KUKA KRL program: MyProgram_109().src

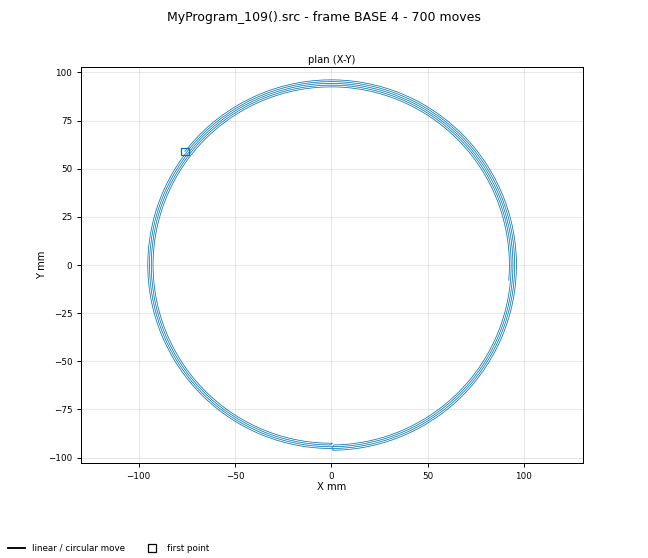
[picture p0: tool path of MyProgram_109().src in frame BASE 4, 700 of 700 moves have a stored position in this frame; points joined in program order, loops and branches not executed]
&ACCESS RVP
&REL 1
&PARAM TEMPLATE = C:\KRC\Roboter\Template\vorgabe
&PARAM EDITMASK = *
DEF MyProgram_109()
; ---- Setting reference (Base) ----
$BASE = BASE_DATA[4]

; --------------------------
; ---- Setting tool (TCP) ----
$TOOL = TOOL_DATA[3]
; --------------------------

$VEL.CP = VEL_APROX_PRINT
Startdeposition()
$VEL.CP = VEL_PRINT
LIN {X -75.9635,Y 58.9825,Z 96,A 136.7179,B 24.9196,C -2.0702,E1 24.8745,E2 -51.4268} C_DIS
LIN {X -71.624,Y 64.1816,Z 96,A 131.6242,B 24.9214,C -2.047,E1 24.884,E2 -46.2546} C_DIS
LIN {X -67.7687,Y 68.2403,Z 96,A 129.5352,B 24.9177,C -2.0948,E1 24.8879,E2 -44.2707} C_DIS
LIN {X -63.6529,Y 72.0961,Z 96,A 126.1542,B 24.9171,C -2.1019,E1 24.8948,E2 -40.8928} C_DIS
LIN {X -60.8353,Y 74.488,Z 96,A 123.6334,B 24.9176,C -2.0964,E1 24.9002,E2 -38.3493} C_DIS
LIN {X -56.4645,Y 77.852,Z 96,A 120.304,B 24.9171,C -2.1019,E1 24.9076,E2 -35.021} C_DIS
LIN {X -51.644,Y 81.1313,Z 96,A 116.9295,B 24.9164,C -2.1118,E1 24.9155,E2 -31.659} C_DIS
LIN {X -49.5866,Y 82.4052,Z 96,A 114.7873,B 24.918,C -2.0916,E1 24.9207,E2 -29.4622} C_DIS
LIN {X -45.8465,Y 84.5421,Z 96,A 112.8787,B 24.9159,C -2.1175,E1 24.9253,E2 -27.6098} C_DIS
LIN {X -39.8443,Y 87.5319,Z 96,A 108.9645,B 24.9152,C -2.1264,E1 24.9351,E2 -23.7067} C_DIS
LIN {X -36.8225,Y 88.8463,Z 96,A 106.6234,B 24.916,C -2.1167,E1 24.9412,E2 -21.337} C_DIS
LIN {X -32.9991,Y 90.3345,Z 96,A 104.4246,B 24.9151,C -2.1281,E1 24.9468,E2 -19.1608} C_DIS
LIN {X -29.4819,Y 91.5429,Z 96,A 101.6282,B 24.9164,C -2.1114,E1 24.9544,E2 -16.3196} C_DIS
LIN {X -25.5098,Y 92.7293,Z 96,A 100.0399,B 24.9138,C -2.1435,E1 24.9585,E2 -14.805} C_DIS
LIN {X -20.1495,Y 94.0393,Z 96,A 96.4801,B 24.9143,C -2.1373,E1 24.9682,E2 -11.2257} C_DIS
LIN {X -16.8432,Y 94.6869,Z 96,A 93.9105,B 24.9157,C -2.1199,E1 24.9754,E2 -8.6122} C_DIS
LIN {X -12.9376,Y 95.3007,Z 96,A 92.2981,B 24.9136,C -2.1465,E1 24.9797,E2 -7.0617} C_DIS
LIN {X -9.0125,Y 95.7501,Z 96,A 89.8172,B 24.9138,C -2.1435,E1 24.9866,E2 -4.5721} C_DIS
LIN {X -5.6055,Y 96.0101,Z 96,A 87.7986,B 24.9138,C -2.1449,E1 24.9922,E2 -2.5561} C_DIS
LIN {X -3.2117,Y 96.1198,Z 96,A 85.5461,B 24.9159,C -2.1171,E1 24.9987,E2 -0.2373} C_DIS
LIN {X 1.3526,Y 96.1645,Z 96,A 83.5892,B 24.9138,C -2.1437,E1 25.0039,E2 1.6563} C_DIS
LIN {X 4.7623,Y 96.0567,Z 96,A 81.5003,B 24.914,C -2.1419,E1 25.0098,E2 3.749} C_DIS
LIN {X 8.4191,Y 95.8048,Z 96,A 79.3633,B 24.9138,C -2.1434,E1 25.0157,E2 5.8814} C_DIS
LIN {X 11.8183,Y 95.4458,Z 96,A 77.2973,B 24.9139,C -2.142,E1 25.0214,E2 7.9492} C_DIS
LIN {X 15.3543,Y 94.9409,Z 96,A 75.1985,B 24.9139,C -2.1424,E1 25.0272,E2 10.045} C_DIS
LIN {X 19.7138,Y 94.1317,Z 96,A 72.7441,B 24.9135,C -2.1479,E1 25.0339,E2 12.4835} C_DIS
LIN {X 25.2917,Y 92.7882,Z 96,A 69.3515,B 24.9135,C -2.1468,E1 25.0431,E2 15.8737} C_DIS
LIN {X 29.6089,Y 91.5018,Z 96,A 66.6503,B 24.9138,C -2.1442,E1 25.0503,E2 18.5764} C_DIS
LIN {X 32.7031,Y 90.4425,Z 96,A 64.5541,B 24.9143,C -2.1372,E1 25.0559,E2 20.6849} C_DIS
LIN {X 35.084,Y 89.5455,Z 96,A 62.7776,B 24.9152,C -2.1264,E1 25.0606,E2 22.4831} C_DIS
LIN {X 40.332,Y 87.3079,Z 96,A 59.687,B 24.9146,C -2.1337,E1 25.0684,E2 25.5489} C_DIS
LIN {X 43.239,Y 85.9067,Z 96,A 57.7408,B 24.9149,C -2.1304,E1 25.0733,E2 27.4977} C_DIS
LIN {X 45.9132,Y 84.5059,Z 96,A 55.8586,B 24.9153,C -2.125,E1 25.0779,E2 29.3873} C_DIS
LIN {X 49.0395,Y 82.731,Z 96,A 53.7927,B 24.9153,C -2.1246,E1 25.0829,E2 31.4477} C_DIS
LIN {X 53.5705,Y 79.8712,Z 96,A 50.4819,B 24.9161,C -2.1153,E1 25.0907,E2 34.7699} C_DIS
LIN {X 56.5092,Y 77.8211,Z 96,A 48.2139,B 24.9168,C -2.1068,E1 25.0959,E2 37.0501} C_DIS
LIN {X 60.8788,Y 74.4528,Z 96,A 45.1605,B 24.9166,C -2.1093,E1 25.1025,E2 40.0861} C_DIS
LIN {X 66.2445,Y 69.7221,Z 96,A 40.9352,B 24.9171,C -2.1021,E1 25.1113,E2 44.3115} C_DIS
LIN {X 68.9933,Y 67.0025,Z 96,A 38.1075,B 24.919,C -2.0778,E1 25.1169,E2 47.1846} C_DIS
LIN {X 71.5664,Y 64.2459,Z 96,A 36.4875,B 24.9176,C -2.096,E1 25.1199,E2 48.7544} C_DIS
LIN {X 73.2967,Y 62.2647,Z 96,A 34.5911,B 24.9189,C -2.0801,E1 25.1234,E2 50.6797} C_DIS
LIN {X 75.914,Y 59.0468,Z 96,A 32.1059,B 24.9194,C -2.0737,E1 25.1277,E2 53.1686} C_DIS
LIN {X 78.5859,Y 55.4417,Z 96,A 29.6936,B 24.9191,C -2.0768,E1 25.1316,E2 55.5618} C_DIS
LIN {X 80.5905,Y 52.4835,Z 96,A 27.4533,B 24.9199,C -2.0671,E1 25.1351,E2 57.8137} C_DIS
LIN {X 82.391,Y 49.6099,Z 96,A 25.7028,B 24.9195,C -2.072,E1 25.1376,E2 59.5439} C_DIS
LIN {X 85.0356,Y 44.9247,Z 96,A 22.1086,B 24.9213,C -2.0486,E1 25.1425,E2 63.1744} C_DIS
LIN {X 87.1678,Y 40.6331,Z 96,A 19.8069,B 24.9203,C -2.0615,E1 25.1452,E2 65.4332} C_DIS
LIN {X 89.0887,Y 36.2281,Z 96,A 16.8208,B 24.9213,C -2.0486,E1 25.1485,E2 68.4335} C_DIS
LIN {X 90.7833,Y 31.7437,Z 96,A 13.9291,B 24.9221,C -2.0388,E1 25.1513,E2 71.3321} C_DIS
LIN {X 92.5603,Y 26.1125,Z 96,A 10.452,B 24.9227,C -2.0298,E1 25.1542,E2 74.8108} C_DIS
LIN {X 93.3092,Y 23.301,Z 96,A 8.1375,B 24.9248,C -2.0023,E1 25.1558,E2 77.1767} C_DIS
LIN {X 94.1518,Y 19.6159,Z 96,A 6.4875,B 24.9236,C -2.0183,E1 25.1567,E2 78.7795} C_DIS
LIN {X 94.8044,Y 16.171,Z 96,A 4.4178,B 24.9241,C -2.0125,E1 25.1577,E2 80.8507} C_DIS
LIN {X 95.3297,Y 12.7141,Z 96,A 2.338,B 24.9245,C -2.006,E1 25.1586,E2 82.9335} C_DIS
LIN {X 95.7187,Y 9.3522,Z 96,A 0.2659,B 24.9252,C -1.9975,E1 25.1592,E2 85.0135} C_DIS
LIN {X 96.0088,Y 5.6288,Z 96,A -1.8781,B 24.9255,C -1.9935,E1 25.1596,E2 87.1542} C_DIS
LIN {X 96.1411,Y 2.5178,Z 96,A -3.7568,B 24.926,C -1.9866,E1 25.1598,E2 89.0379} C_DIS
LIN {X 96.1691,Y -0.9828,Z 96,A -5.8078,B 24.9264,C -1.9813,E1 25.1598,E2 91.0894} C_DIS
LIN {X 96.0512,Y -4.8615,Z 96,A -8.2755,B 24.9274,C -1.9678,E1 25.1595,E2 93.5741} C_DIS
LIN {X 95.7693,Y -8.8044,Z 96,A -10.4034,B 24.9274,C -1.969,E1 25.159,E2 95.6867} C_DIS
LIN {X 95.3701,Y -12.4021,Z 96,A -12.583,B 24.9279,C -1.9611,E1 25.1583,E2 97.8719} C_DIS
LIN {X 94.8345,Y -15.991,Z 96,A -14.5993,B 24.9279,C -1.9598,E1 25.1574,E2 99.8795} C_DIS
LIN {X 94.3756,Y -18.5099,Z 96,A -16.6489,B 24.9298,C -1.9348,E1 25.1563,E2 101.9762} C_DIS
LIN {X 93.7019,Y -21.6617,Z 96,A -18.0886,B 24.9289,C -1.9471,E1 25.1554,E2 103.3784} C_DIS
LIN {X 93.134,Y -23.986,Z 96,A -20.0266,B 24.9307,C -1.9229,E1 25.154,E2 105.3622} C_DIS
LIN {X 92.2114,Y -27.3189,Z 96,A -22.127,B 24.9313,C -1.9149,E1 25.1524,E2 107.4695} C_DIS
LIN {X 91.1057,Y -30.8062,Z 96,A -23.3453,B 24.9291,C -1.945,E1 25.1514,E2 108.61} C_DIS
LIN {X 89.8798,Y -34.2186,Z 96,A -26.3157,B 24.9318,C -1.9072,E1 25.1484,E2 111.653} C_DIS
LIN {X 88.6877,Y -37.1993,Z 96,A -28.0731,B 24.9318,C -1.9072,E1 25.1465,E2 113.4006} C_DIS
LIN {X 86.7733,Y -41.4693,Z 96,A -30.9801,B 24.9327,C -1.8943,E1 25.1431,E2 116.3224} C_DIS
LIN {X 85.3222,Y -44.3806,Z 96,A -32.8135,B 24.9329,C -1.8925,E1 25.1408,E2 118.1503} C_DIS
LIN {X 81.7409,Y -50.6735,Z 96,A -36.7914,B 24.9329,C -1.8929,E1 25.1352,E2 122.1068} C_DIS
LIN {X 79.0751,Y -54.7396,Z 96,A -39.9312,B 24.9341,C -1.8755,E1 25.1303,E2 125.2721} C_DIS
LIN {X 75.347,Y -59.7672,Z 96,A -43.4414,B 24.9341,C -1.8738,E1 25.1243,E2 128.7697} C_DIS
LIN {X 73.0047,Y -62.6074,Z 96,A -45.4134,B 24.934,C -1.8765,E1 25.1208,E2 130.7263} C_DIS
LIN {X 70.1761,Y -65.7618,Z 96,A -48.3985,B 24.9357,C -1.8527,E1 25.1151,E2 133.7545} C_DIS
LIN {X 66.9268,Y -69.0661,Z 96,A -50.7849,B 24.9351,C -1.8601,E1 25.1105,E2 136.1133} C_DIS
LIN {X 64.5588,Y -71.2861,Z 96,A -52.5649,B 24.9351,C -1.8613,E1 25.1068,E2 137.8831} C_DIS
LIN {X 61.8693,Y -73.6324,Z 96,A -55.2908,B 24.937,C -1.834,E1 25.1009,E2 140.663} C_DIS
LIN {X 59.3273,Y -75.6948,Z 96,A -56.8127,B 24.9361,C -1.8458,E1 25.0977,E2 142.1513} C_DIS
LIN {X 56.7069,Y -77.6763,Z 96,A -58.7892,B 24.9365,C -1.841,E1 25.0932,E2 144.1322} C_DIS
LIN {X 54.6408,Y -79.1438,Z 96,A -60.489,B 24.9372,C -1.8308,E1 25.0893,E2 145.8502} C_DIS
LIN {X 48.4141,Y -83.1004,Z 96,A -64.6992,B 24.9372,C -1.8294,E1 25.0793,E2 150.0504} C_DIS
LIN {X 43.3453,Y -85.8526,Z 96,A -68.4345,B 24.9384,C -1.8125,E1 25.07,E2 153.8152} C_DIS
LIN {X 38.7385,Y -88.0268,Z 96,A -70.8505,B 24.9372,C -1.8306,E1 25.064,E2 156.1822} C_DIS
LIN {X 36.2891,Y -89.0639,Z 96,A -72.9477,B 24.9386,C -1.8095,E1 25.0585,E2 158.3245} C_DIS
LIN {X 32.3499,Y -90.5704,Z 96,A -76.1015,B 24.9404,C -1.7829,E1 25.0501,E2 161.5346} C_DIS
LIN {X 27.4941,Y -92.1595,Z 96,A -77.8804,B 24.9376,C -1.8253,E1 25.0456,E2 163.2102} C_DIS
LIN {X 22.4848,Y -93.5083,Z 96,A -81.358,B 24.9387,C -1.8079,E1 25.0361,E2 166.7234} C_DIS
LIN {X 17.5814,Y -94.5541,Z 96,A -84.3174,B 24.9388,C -1.8063,E1 25.028,E2 169.6831} C_DIS
LIN {X 14.1878,Y -95.1222,Z 96,A -86.3586,B 24.9389,C -1.8051,E1 25.0223,E2 171.725} C_DIS
LIN {X 10.552,Y -95.594,Z 96,A -88.5213,B 24.9389,C -1.8045,E1 25.0163,E2 173.8875} C_DIS
LIN {X 7.0264,Y -95.9176,Z 96,A -90.6506,B 24.9391,C -1.8028,E1 25.0104,E2 176.0198} C_DIS
LIN {X 3.4991,Y -96.111,Z 96,A -92.7507,B 24.9391,C -1.8022,E1 25.0046,E2 178.1207} C_DIS
LIN {X 0.6665,Y -96.1682,Z 96,A -93.7382,B 24.9374,C -1.8268,E1 25.002,E2 179.0497} C_DIS
Enddeposition()
LIN {X 0.6665,Y -96.1682,Z 96,A -93.7382,B 24.9374,C -1.8268,E1 25.002,E2 179.0497} C_DIS
Startdeposition()
$VEL.CP = VEL_PRINT
LIN {X 1.0872,Y -95.2543,Z 96,A -93.1803,B 24.9356,C -1.8535,E1 25.0037,E2 178.4284} C_DIS
LIN {X 4.3828,Y -95.1587,Z 96,A -91.1856,B 24.9356,C -1.8547,E1 25.0093,E2 176.4315} C_DIS
LIN {X 7.8747,Y -94.9336,Z 96,A -89.0988,B 24.9355,C -1.855,E1 25.0151,E2 174.3449} C_DIS
LIN {X 11.567,Y -94.5556,Z 96,A -86.7396,B 24.9351,C -1.8609,E1 25.0217,E2 171.9734} C_DIS
LIN {X 15.6874,Y -93.9586,Z 96,A -84.4427,B 24.9355,C -1.8552,E1 25.028,E2 169.6922} C_DIS
LIN {X 21.2338,Y -92.8627,Z 96,A -81.221,B 24.9357,C -1.8516,E1 25.0367,E2 166.483} C_DIS
LIN {X 24.7928,Y -91.9762,Z 96,A -78.7965,B 24.935,C -1.8619,E1 25.0433,E2 164.038} C_DIS
LIN {X 28.3124,Y -90.9545,Z 96,A -76.1297,B 24.9336,C -1.8815,E1 25.0506,E2 161.3294} C_DIS
LIN {X 31.5787,Y -89.8727,Z 96,A -74.2994,B 24.9341,C -1.8753,E1 25.0554,E2 159.5176} C_DIS
LIN {X 37.2004,Y -87.6954,Z 96,A -71.1813,B 24.935,C -1.8615,E1 25.0633,E2 156.439} C_DIS
LIN {X 39.5771,Y -86.6498,Z 96,A -69.4286,B 24.9344,C -1.871,E1 25.0679,E2 154.6683} C_DIS
LIN {X 42.7302,Y -85.1391,Z 96,A -66.5179,B 24.932,C -1.9047,E1 25.0753,E2 151.6857} C_DIS
LIN {X 46.6327,Y -83.0647,Z 96,A -64.7132,B 24.9339,C -1.8773,E1 25.0796,E2 149.9511} C_DIS
LIN {X 49.7001,Y -81.2667,Z 96,A -62.137,B 24.9325,C -1.8977,E1 25.0858,E2 147.3347} C_DIS
LIN {X 55.4137,Y -77.4831,Z 96,A -58.4667,B 24.9331,C -1.8888,E1 25.0942,E2 143.6976} C_DIS
LIN {X 58.1709,Y -75.4351,Z 96,A -55.6801,B 24.9308,C -1.9206,E1 25.1005,E2 140.8461} C_DIS
LIN {X 61.4032,Y -72.8299,Z 96,A -53.3642,B 24.9309,C -1.9193,E1 25.1054,E2 138.5423} C_DIS
LIN {X 64.027,Y -70.5345,Z 96,A -51.9557,B 24.9325,C -1.8979,E1 25.1083,E2 137.1899} C_DIS
LIN {X 65.8828,Y -68.8031,Z 96,A -50.2594,B 24.9318,C -1.908,E1 25.1117,E2 135.4768} C_DIS
LIN {X 69.6881,Y -64.9467,Z 96,A -46.334,B 24.9293,C -1.9416,E1 25.1194,E2 131.489} C_DIS
LIN {X 72.4219,Y -61.8822,Z 96,A -44.6671,B 24.9311,C -1.9171,E1 25.1224,E2 129.8874} C_DIS
LIN {X 74.3382,Y -59.5687,Z 96,A -41.9522,B 24.9282,C -1.9569,E1 25.1273,E2 127.0913} C_DIS
LIN {X 77.1265,Y -55.9108,Z 96,A -39.576,B 24.9288,C -1.9493,E1 25.1311,E2 124.7444} C_DIS
LIN {X 80.3004,Y -51.2466,Z 96,A -36.6114,B 24.9293,C -1.9423,E1 25.1356,E2 121.8112} C_DIS
LIN {X 83.327,Y -46.163,Z 96,A -33.0482,B 24.9285,C -1.9527,E1 25.1406,E2 118.2418} C_DIS
LIN {X 85.4364,Y -42.1302,Z 96,A -30.4276,B 24.9282,C -1.9563,E1 25.144,E2 115.6265} C_DIS
LIN {X 87.4708,Y -37.7268,Z 96,A -27.6993,B 24.9282,C -1.9578,E1 25.1471,E2 112.9095} C_DIS
LIN {X 89.7057,Y -32.0544,Z 96,A -23.7893,B 24.9266,C -1.9784,E1 25.1511,E2 108.9726} C_DIS
LIN {X 90.7958,Y -28.8219,Z 96,A -20.9247,B 24.9238,C -2.0165,E1 25.1535,E2 106.0343} C_DIS
LIN {X 92.1449,Y -24.163,Z 96,A -19.1061,B 24.9263,C -1.9829,E1 25.1548,E2 104.3054} C_DIS
LIN {X 92.8385,Y -21.3386,Z 96,A -16.7169,B 24.924,C -2.0134,E1 25.1564,E2 101.8583} C_DIS
LIN {X 93.524,Y -18.0992,Z 96,A -15.4794,B 24.9257,C -1.9905,E1 25.157,E2 100.6821} C_DIS
LIN {X 93.95,Y -15.7388,Z 96,A -13.7684,B 24.9246,C -2.0055,E1 25.1578,E2 98.9457} C_DIS
LIN {X 94.4624,Y -12.2949,Z 96,A -11.7086,B 24.9242,C -2.0109,E1 25.1586,E2 96.8854} C_DIS
LIN {X 94.8478,Y -8.8439,Z 96,A -9.6239,B 24.9237,C -2.0174,E1 25.1592,E2 94.7975} C_DIS
LIN {X 95.1282,Y -4.9993,Z 96,A -7.3977,B 24.9234,C -2.0213,E1 25.1596,E2 92.5753} C_DIS
LIN {X 95.2462,Y -1.5801,Z 96,A -5.2259,B 24.9225,C -2.0324,E1 25.1598,E2 90.3904} C_DIS
LIN {X 95.2392,Y 1.9593,Z 96,A -3.1527,B 24.9222,C -2.037,E1 25.1598,E2 88.3184} C_DIS
LIN {X 95.1078,Y 5.3688,Z 96,A -1.1401,B 24.9218,C -2.0421,E1 25.1594,E2 86.3059} C_DIS
LIN {X 94.8541,Y 8.7756,Z 96,A 0.9363,B 24.9212,C -2.0495,E1 25.159,E2 84.2244} C_DIS
LIN {X 94.4613,Y 12.3033,Z 96,A 3.0514,B 24.9208,C -2.0555,E1 25.1583,E2 82.1077} C_DIS
LIN {X 93.918,Y 15.9302,Z 96,A 5.3098,B 24.9201,C -2.0644,E1 25.1573,E2 79.8414} C_DIS
LIN {X 93.2612,Y 19.4094,Z 96,A 8.2612,B 24.9171,C -2.1029,E1 25.1556,E2 76.8164} C_DIS
LIN {X 92.1175,Y 24.2694,Z 96,A 10.2054,B 24.9196,C -2.0711,E1 25.1543,E2 74.9585} C_DIS
LIN {X 91.0329,Y 28.0596,Z 96,A 12.9347,B 24.9179,C -2.092,E1 25.1521,E2 72.1954} C_DIS
LIN {X 88.9459,Y 34.104,Z 96,A 16.6021,B 24.9176,C -2.0965,E1 25.1486,E2 68.538} C_DIS
LIN {X 87.6252,Y 37.3672,Z 96,A 18.876,B 24.9166,C -2.1086,E1 25.1462,E2 66.248} C_DIS
LIN {X 85.6149,Y 41.7698,Z 96,A 22.096,B 24.915,C -2.1286,E1 25.1423,E2 62.9981} C_DIS
LIN {X 83.9203,Y 45.076,Z 96,A 23.6557,B 24.9166,C -2.1089,E1 25.1403,E2 61.4931} C_DIS
LIN {X 81.7775,Y 48.8564,Z 96,A 26.1789,B 24.9163,C -2.1125,E1 25.1368,E2 58.9744} C_DIS
LIN {X 80.3931,Y 51.1021,Z 96,A 28.2852,B 24.9144,C -2.1364,E1 25.1336,E2 56.8225} C_DIS
LIN {X 77.954,Y 54.7513,Z 96,A 30.614,B 24.9148,C -2.1312,E1 25.1299,E2 54.5172} C_DIS
LIN {X 74.8472,Y 58.9257,Z 96,A 34.1679,B 24.9129,C -2.1549,E1 25.1238,E2 50.9243} C_DIS
LIN {X 72.6176,Y 61.6524,Z 96,A 35.6693,B 24.9144,C -2.1365,E1 25.1212,E2 49.4731} C_DIS
LIN {X 70.5715,Y 63.9867,Z 96,A 38.272,B 24.9118,C -2.1684,E1 25.1162,E2 46.8066} C_DIS
LIN {X 67.8593,Y 66.8538,Z 96,A 39.8824,B 24.9137,C -2.1449,E1 25.1132,E2 45.2587} C_DIS
LIN {X 65.328,Y 69.3294,Z 96,A 42.9783,B 24.9104,C -2.1855,E1 25.1068,E2 42.0795} C_DIS
LIN {X 61.7288,Y 72.5525,Z 96,A 44.9914,B 24.9127,C -2.1577,E1 25.1027,E2 40.14} C_DIS
LIN {X 58.2198,Y 75.3975,Z 96,A 47.2958,B 24.9135,C -2.1475,E1 25.0977,E2 37.8685} C_DIS
LIN {X 55.7027,Y 77.277,Z 96,A 49.5726,B 24.9121,C -2.165,E1 25.0925,E2 35.5583} C_DIS
LIN {X 50.921,Y 80.5087,Z 96,A 52.8806,B 24.9121,C -2.1646,E1 25.0849,E2 32.2624} C_DIS
LIN {X 47.3722,Y 82.645,Z 96,A 55.4654,B 24.9115,C -2.1717,E1 25.0786,E2 29.6687} C_DIS
LIN {X 44.2239,Y 84.3717,Z 96,A 57.403,B 24.912,C -2.1665,E1 25.0739,E2 27.749} C_DIS
LIN {X 42.1748,Y 85.4144,Z 96,A 59.1206,B 24.9108,C -2.1804,E1 25.0695,E2 26.0031} C_DIS
LIN {X 38.4057,Y 87.1748,Z 96,A 62.1578,B 24.909,C -2.2027,E1 25.0617,E2 22.9206} C_DIS
LIN {X 34.9011,Y 88.6354,Z 96,A 63.5697,B 24.9114,C -2.1735,E1 25.0582,E2 21.5811} C_DIS
LIN {X 32.6409,Y 89.4923,Z 96,A 65.2605,B 24.9106,C -2.1834,E1 25.0537,E2 19.8705} C_DIS
LIN {X 28.8125,Y 90.7989,Z 96,A 68.2218,B 24.9089,C -2.2043,E1 25.0458,E2 16.8652} C_DIS
LIN {X 25.4772,Y 91.7904,Z 96,A 69.6449,B 24.9107,C -2.1817,E1 25.0421,E2 15.4979} C_DIS
LIN {X 23.1402,Y 92.4072,Z 96,A 71.7537,B 24.9087,C -2.206,E1 25.0362,E2 13.3348} C_DIS
LIN {X 19.7611,Y 93.1886,Z 96,A 73.6606,B 24.9092,C -2.2006,E1 25.0311,E2 11.4432} C_DIS
LIN {X 16.0236,Y 93.9024,Z 96,A 75.5551,B 24.9102,C -2.1875,E1 25.026,E2 9.5818} C_DIS
LIN {X 13.1162,Y 94.3523,Z 96,A 77.4705,B 24.9098,C -2.1931,E1 25.0206,E2 7.6548} C_DIS
LIN {X 9.6502,Y 94.7695,Z 96,A 79.4669,B 24.9101,C -2.1898,E1 25.0151,E2 5.6677} C_DIS
LIN {X 6.4585,Y 95.04,Z 96,A 81.3482,B 24.9101,C -2.1883,E1 25.0099,E2 3.7908} C_DIS
LIN {X 3.128,Y 95.208,Z 96,A 83.3988,B 24.9101,C -2.1898,E1 25.0042,E2 1.7374} C_DIS
LIN {X -0.1984,Y 95.2593,Z 96,A 85.7914,B 24.909,C -2.203,E1 24.9974,E2 -0.6866} C_DIS
LIN {X -5.0768,Y 95.124,Z 96,A 88.3402,B 24.9101,C -2.1887,E1 24.9904,E2 -3.2017} C_DIS
LIN {X -8.2975,Y 94.8982,Z 96,A 91.1194,B 24.9078,C -2.2168,E1 24.9825,E2 -6.0491} C_DIS
LIN {X -12.8562,Y 94.3892,Z 96,A 92.9174,B 24.9107,C -2.1819,E1 24.9777,E2 -7.7656} C_DIS
LIN {X -18.277,Y 93.4898,Z 96,A 96.3114,B 24.9107,C -2.1825,E1 24.9684,E2 -11.1642} C_DIS
LIN {X -22.9547,Y 92.4528,Z 96,A 99.344,B 24.9105,C -2.1849,E1 24.9601,E2 -14.2066} C_DIS
LIN {X -25.6453,Y 91.7428,Z 96,A 101.5323,B 24.9092,C -2.2007,E1 24.9541,E2 -16.4359} C_DIS
LIN {X -29.2113,Y 90.6699,Z 96,A 102.9294,B 24.9117,C -2.1696,E1 24.9506,E2 -17.7615} C_DIS
LIN {X -31.5975,Y 89.8661,Z 96,A 104.6823,B 24.9112,C -2.1757,E1 24.9459,E2 -19.5324} C_DIS
LIN {X -34.6764,Y 88.7237,Z 96,A 106.9992,B 24.9105,C -2.1846,E1 24.9398,E2 -21.8752} C_DIS
LIN {X -38.9999,Y 86.91,Z 96,A 110.3805,B 24.9093,C -2.1994,E1 24.931,E2 -25.2997} C_DIS
LIN {X -43.2642,Y 84.8677,Z 96,A 112.3516,B 24.912,C -2.1655,E1 24.9263,E2 -27.1955} C_DIS
LIN {X -48.942,Y 81.7269,Z 96,A 116.0651,B 24.9131,C -2.1524,E1 24.9173,E2 -30.8885} C_DIS
LIN {X -51.9423,Y 79.8527,Z 96,A 118.6277,B 24.9123,C -2.1627,E1 24.9112,E2 -33.4839} C_DIS
LIN {X -57.0114,Y 76.3154,Z 96,A 122.1932,B 24.9133,C -2.1501,E1 24.9031,E2 -37.0318} C_DIS
LIN {X -59.6988,Y 74.2327,Z 96,A 124.9562,B 24.9117,C -2.1693,E1 24.897,E2 -39.8509} C_DIS
LIN {X -62.9852,Y 71.4658,Z 96,A 127.6584,B 24.9119,C -2.1674,E1 24.8913,E2 -42.5592} C_DIS
LIN {X -66.4029,Y 68.3018,Z 96,A 129.6912,B 24.9145,C -2.1355,E1 24.8873,E2 -44.5245} C_DIS
LIN {X -71.0089,Y 63.4984,Z 96,A 134.2396,B 24.9138,C -2.1434,E1 24.8786,E2 -49.1115} C_DIS
LIN {X -73.4528,Y 60.6554,Z 96,A 135.7348,B 24.9163,C -2.1129,E1 24.8761,E2 -50.5409} C_DIS
LIN {X -74.9969,Y 58.7363,Z 96,A 137.5717,B 24.9157,C -2.1204,E1 24.8728,E2 -52.4044} C_DIS
LIN {X -77.9953,Y 54.6919,Z 96,A 140.4948,B 24.9166,C -2.1088,E1 24.8681,E2 -55.314} C_DIS
LIN {X -80.3638,Y 51.1478,Z 96,A 142.9077,B 24.9175,C -2.0968,E1 24.8644,E2 -57.7104} C_DIS
LIN {X -81.5228,Y 49.2788,Z 96,A 144.8947,B 24.9162,C -2.1144,E1 24.8615,E2 -59.7496} C_DIS
LIN {X -83.282,Y 46.2435,Z 96,A 146.3012,B 24.9184,C -2.0857,E1 24.8596,E2 -61.095} C_DIS
LIN {X -85.6489,Y 41.6961,Z 96,A 149.6025,B 24.9186,C -2.0835,E1 24.8554,E2 -64.4088} C_DIS
LIN {X -87.122,Y 38.5268,Z 96,A 152.1913,B 24.9179,C -2.0927,E1 24.8524,E2 -67.0339} C_DIS
LIN {X -88.4184,Y 35.4506,Z 96,A 153.7568,B 24.9195,C -2.0725,E1 24.8508,E2 -68.5596} C_DIS
LIN {X -89.9884,Y 31.2488,Z 96,A 156.3114,B 24.9205,C -2.0596,E1 24.8484,E2 -71.098} C_DIS
LIN {X -90.9272,Y 28.4006,Z 96,A 158.8014,B 24.9192,C -2.0759,E1 24.8462,E2 -73.6411} C_DIS
LIN {X -91.9184,Y 25.007,Z 96,A 160.8116,B 24.92,C -2.0654,E1 24.8448,E2 -75.6381} C_DIS
LIN {X -92.8299,Y 21.3756,Z 96,A 163.0358,B 24.9206,C -2.0574,E1 24.8434,E2 -77.8562} C_DIS
LIN {X -94.0127,Y 15.3638,Z 96,A 167.6057,B 24.9193,C -2.0741,E1 24.8412,E2 -82.4931} C_DIS
LIN {X -94.7949,Y 9.4075,Z 96,A 169.84,B 24.9236,C -2.0182,E1 24.8405,E2 -84.6074} C_DIS
LIN {X -95.1699,Y 4.1221,Z 96,A 173.7598,B 24.9226,C -2.0313,E1 24.8398,E2 -88.582} C_DIS
LIN {X -95.2578,Y 0.6008,Z 96,A 175.2863,B 24.9246,C -2.0056,E1 24.8398,E2 -90.0563} C_DIS
LIN {X -95.2219,Y -2.6748,Z 96,A 177.9803,B 24.9233,C -2.0224,E1 24.84,E2 -92.8067} C_DIS
LIN {X -95.036,Y -6.5179,Z 96,A -179.7635,B 24.924,C -2.0132,E1 24.8404,E2 -95.0544} C_DIS
LIN {X -94.7217,Y -10.1067,Z 96,A -178.3175,B 24.9263,C -1.9832,E1 24.8408,E2 -96.4376} C_DIS
LIN {X -94.3898,Y -12.8522,Z 96,A -175.5181,B 24.9239,C -2.0144,E1 24.8419,E2 -99.3283} C_DIS
LIN {X -93.5955,Y -17.7279,Z 96,A -172.6319,B 24.9248,C -2.0024,E1 24.8434,E2 -102.2029} C_DIS
LIN {X -92.6273,Y -22.2399,Z 96,A -170.6522,B 24.9274,C -1.9682,E1 24.8446,E2 -104.1125} C_DIS
LIN {X -91.7533,Y -25.6082,Z 96,A -167.8083,B 24.926,C -1.9861,E1 24.8468,E2 -107.0156} C_DIS
LIN {X -90.4912,Y -29.7636,Z 96,A -166.119,B 24.9288,C -1.9485,E1 24.8481,E2 -108.6248} C_DIS
LIN {X -89.0865,Y -33.7328,Z 96,A -162.7865,B 24.9275,C -1.9669,E1 24.8514,E2 -112.02} C_DIS
LIN {X -87.6764,Y -37.2455,Z 96,A -161.1154,B 24.9294,C -1.9407,E1 24.8531,E2 -113.6379} C_DIS
LIN {X -86.8228,Y -39.1933,Z 96,A -159.4056,B 24.9286,C -1.951,E1 24.8551,E2 -115.3817} C_DIS
LIN {X -83.3712,Y -46.0839,Z 96,A -155.3646,B 24.931,C -1.9189,E1 24.8602,E2 -119.3677} C_DIS
LIN {X -81.4344,Y -49.4242,Z 96,A -152.8186,B 24.9309,C -1.92,E1 24.8639,E2 -121.9295} C_DIS
LIN {X -80.0366,Y -51.6576,Z 96,A -151.1272,B 24.9309,C -1.9194,E1 24.8664,E2 -123.6279} C_DIS
LIN {X -77.5633,Y -55.3014,Z 96,A -148.2247,B 24.9309,C -1.921,E1 24.8711,E2 -126.5488} C_DIS
LIN {X -74.8125,Y -58.9695,Z 96,A -145.887,B 24.9323,C -1.9006,E1 24.875,E2 -128.8488} C_DIS
LIN {X -73.1049,Y -61.0741,Z 96,A -143.2197,B 24.9301,C -1.9312,E1 24.8799,E2 -131.6012} C_DIS
LIN {X -69.8305,Y -64.7943,Z 96,A -141.0485,B 24.9325,C -1.8975,E1 24.8839,E2 -133.7019} C_DIS
LIN {X -67.4187,Y -67.2999,Z 96,A -138.4075,B 24.9315,C -1.9114,E1 24.8892,E2 -136.3872} C_DIS
LIN {X -64.6426,Y -69.9696,Z 96,A -136.9837,B 24.934,C -1.8769,E1 24.8919,E2 -137.7347} C_DIS
LIN {X -60.9411,Y -73.2154,Z 96,A -133.7522,B 24.9337,C -1.8802,E1 24.8988,E2 -140.9866} C_DIS
LIN {X -57.9716,Y -75.5887,Z 96,A -131.5799,B 24.9343,C -1.8722,E1 24.9035,E2 -143.148} C_DIS
LIN {X -54.2195,Y -78.3236,Z 96,A -128.301,B 24.9335,C -1.8839,E1 24.9111,E2 -146.466} C_DIS
LIN {X -50.7684,Y -80.604,Z 96,A -126.153,B 24.9346,C -1.8685,E1 24.916,E2 -148.5843} C_DIS
LIN {X -48.1602,Y -82.189,Z 96,A -124.2715,B 24.9346,C -1.8674,E1 24.9206,E2 -150.469} C_DIS
LIN {X -44.9607,Y -83.9829,Z 96,A -122.0378,B 24.9348,C -1.8654,E1 24.926,E2 -152.7041} C_DIS
LIN {X -41.7501,Y -85.6225,Z 96,A -119.1409,B 24.9332,C -1.8878,E1 24.9335,E2 -155.6621} C_DIS
LIN {X -37.7165,Y -87.4753,Z 96,A -117.6159,B 24.9362,C -1.8455,E1 24.9371,E2 -157.09} C_DIS
LIN {X -34.2101,Y -88.9057,Z 96,A -114.6795,B 24.9347,C -1.8659,E1 24.9449,E2 -160.0813} C_DIS
LIN {X -28.2689,Y -90.968,Z 96,A -111.1811,B 24.9356,C -1.853,E1 24.9541,E2 -163.5556} C_DIS
LIN {X -23.0396,Y -92.4322,Z 96,A -107.6202,B 24.9351,C -1.8612,E1 24.9637,E2 -167.1416} C_DIS
LIN {X -19.7403,Y -93.1931,Z 96,A -105.8008,B 24.9357,C -1.8527,E1 24.9686,E2 -168.9428} C_DIS
LIN {X -16.418,Y -93.8348,Z 96,A -103.7725,B 24.9357,C -1.8517,E1 24.9742,E2 -170.971} C_DIS
LIN {X -13.1715,Y -94.3444,Z 96,A -101.7508,B 24.9357,C -1.8528,E1 24.9798,E2 -172.9971} C_DIS
LIN {X -9.6435,Y -94.7702,Z 96,A -99.6109,B 24.9357,C -1.8527,E1 24.9857,E2 -175.1378} C_DIS
LIN {X -5.8991,Y -95.0778,Z 96,A -97.3638,B 24.9357,C -1.8522,E1 24.992,E2 -177.3847} C_DIS
LIN {X -2.4876,Y -95.2277,Z 96,A -95.3064,B 24.9357,C -1.8526,E1 24.9978,E2 -179.4433} C_DIS
LIN {X 0.6651,Y -95.2549,Z 96,A -94.235,B 24.9377,C -1.8237,E1 25.0006,E2 -180.4464} C_DIS
Enddeposition()
LIN {X 0.6651,Y -95.2549,Z 96,A -94.235,B 24.9377,C -1.8237,E1 25.0006,E2 -180.4464} C_DIS
Startdeposition()
$VEL.CP = VEL_PRINT
LIN {X 0.2729,Y -94.3453,Z 96,A -94.7204,B 24.9372,C -1.831,E1 24.9993,E2 -179.9782} C_DIS
LIN {X -3.2853,Y -94.2888,Z 96,A -96.8702,B 24.9372,C -1.8311,E1 24.9932,E2 -177.8283} C_DIS
LIN {X -6.522,Y -94.1197,Z 96,A -98.8771,B 24.9372,C -1.8297,E1 24.9876,E2 -175.8176} C_DIS
LIN {X -9.9655,Y -93.8175,Z 96,A -100.9241,B 24.9372,C -1.8317,E1 24.982,E2 -173.7741} C_DIS
LIN {X -13.2272,Y -93.4134,Z 96,A -102.8791,B 24.937,C -1.8335,E1 24.9766,E2 -171.8219} C_DIS
LIN {X -16.7128,Y -92.8531,Z 96,A -105.0154,B 24.937,C -1.8344,E1 24.9707,E2 -169.6858} C_DIS
LIN {X -21.4523,Y -91.8742,Z 96,A -107.8471,B 24.9366,C -1.8394,E1 24.963,E2 -166.8624} C_DIS
LIN {X -24.0799,Y -91.2212,Z 96,A -109.7685,B 24.9372,C -1.8309,E1 24.9577,E2 -164.9181} C_DIS
LIN {X -27.8238,Y -90.1492,Z 96,A -111.8106,B 24.9363,C -1.8435,E1 24.9523,E2 -162.9025} C_DIS
LIN {X -31.0447,Y -89.0915,Z 96,A -114.169,B 24.9369,C -1.835,E1 24.946,E2 -160.5196} C_DIS
LIN {X -34.5678,Y -87.7844,Z 96,A -116.2895,B 24.9364,C -1.8426,E1 24.9405,E2 -158.4125} C_DIS
LIN {X -37.4941,Y -86.5752,Z 96,A -119.4711,B 24.9391,C -1.8031,E1 24.9321,E2 -155.1296} C_DIS
LIN {X -42.8069,Y -84.075,Z 96,A -122.2947,B 24.9371,C -1.8317,E1 24.9252,E2 -152.3666} C_DIS
LIN {X -45.6701,Y -82.5554,Z 96,A -123.7498,B 24.9358,C -1.8513,E1 24.9217,E2 -150.9538} C_DIS
LIN {X -48.2436,Y -81.0781,Z 96,A -125.5343,B 24.9355,C -1.8544,E1 24.9174,E2 -149.1714} C_DIS
LIN {X -51.4978,Y -79.0523,Z 96,A -128.5673,B 24.9369,C -1.8349,E1 24.9102,E2 -146.0824} C_DIS
LIN {X -54.5606,Y -76.9691,Z 96,A -130.4376,B 24.9358,C -1.851,E1 24.906,E2 -144.2439} C_DIS
LIN {X -58.058,Y -74.368,Z 96,A -132.9719,B 24.9352,C -1.8593,E1 24.9004,E2 -141.7201} C_DIS
LIN {X -60.7096,Y -72.2194,Z 96,A -135.0933,B 24.935,C -1.8616,E1 24.8958,E2 -139.5962} C_DIS
LIN {X -63.6332,Y -69.6554,Z 96,A -137.7244,B 24.9353,C -1.8576,E1 24.8903,E2 -136.9451} C_DIS
LIN {X -67.1546,Y -66.2668,Z 96,A -140.2784,B 24.9339,C -1.8771,E1 24.8853,E2 -134.4268} C_DIS
LIN {X -69.4973,Y -63.8055,Z 96,A -142.1591,B 24.9332,C -1.8875,E1 24.8817,E2 -132.5627} C_DIS
LIN {X -72.2652,Y -60.6546,Z 96,A -144.9903,B 24.9334,C -1.8842,E1 24.8765,E2 -129.7107} C_DIS
LIN {X -74.0205,Y -58.4977,Z 96,A -146.5759,B 24.9329,C -1.8915,E1 24.8738,E2 -128.135} C_DIS
LIN {X -77.4194,Y -53.9191,Z 96,A -150.2303,B 24.9328,C -1.8939,E1 24.8677,E2 -124.4687} C_DIS
LIN {X -79.4607,Y -50.8628,Z 96,A -152.4591,B 24.9323,C -1.8998,E1 24.8643,E2 -122.2426} C_DIS
LIN {X -81.3228,Y -47.8296,Z 96,A -154.5928,B 24.9319,C -1.9063,E1 24.8613,E2 -120.1136} C_DIS
LIN {X -82.7029,Y -45.4035,Z 96,A -157.4464,B 24.9341,C -1.8749,E1 24.8574,E2 -117.17} C_DIS
LIN {X -85.3496,Y -40.2077,Z 96,A -159.8606,B 24.9309,C -1.9197,E1 24.8545,E2 -114.8496} C_DIS
LIN {X -86.6279,Y -37.3732,Z 96,A -162.4683,B 24.9321,C -1.9028,E1 24.8516,E2 -112.187} C_DIS
LIN {X -88.2211,Y -33.4373,Z 96,A -164.2954,B 24.9299,C -1.9336,E1 24.8498,E2 -110.4232} C_DIS
LIN {X -89.4073,Y -30.1223,Z 96,A -166.2901,B 24.9291,C -1.9444,E1 24.848,E2 -108.4429} C_DIS
LIN {X -90.5858,Y -26.3716,Z 96,A -168.909,B 24.9291,C -1.9444,E1 24.8458,E2 -105.8088} C_DIS
LIN {X -91.411,Y -23.3468,Z 96,A -170.8034,B 24.9287,C -1.9504,E1 24.8445,E2 -103.918} C_DIS
LIN {X -92.5641,Y -18.2506,Z 96,A -173.7598,B 24.9275,C -1.9669,E1 24.8427,E2 -100.9836} C_DIS
LIN {X -93.247,Y -14.3537,Z 96,A -176.6701,B 24.9281,C -1.9588,E1 24.8414,E2 -98.0364} C_DIS
LIN {X -93.705,Y -10.9722,Z 96,A -178.7535,B 24.9276,C -1.965,E1 24.8406,E2 -95.9553} C_DIS
LIN {X -94.1236,Y -6.4644,Z 96,A 178.6146,B 24.9267,C -1.9773,E1 24.8401,E2 -93.3372} C_DIS
LIN {X -94.3318,Y -1.5967,Z 96,A 175.9373,B 24.9253,C -1.9955,E1 24.8398,E2 -90.687} C_DIS
LIN {X -94.263,Y 3.9392,Z 96,A 172.5879,B 24.9245,C -2.0066,E1 24.84,E2 -87.3441} C_DIS
LIN {X -94.0341,Y 7.6565,Z 96,A 170.0379,B 24.9246,C -2.005,E1 24.8404,E2 -84.7749} C_DIS
LIN {X -93.2218,Y 14.5165,Z 96,A 166.0223,B 24.9232,C -2.024,E1 24.8418,E2 -80.7806} C_DIS
LIN {X -92.3038,Y 19.527,Z 96,A 162.6774,B 24.923,C -2.0261,E1 24.8436,E2 -77.4208} C_DIS
LIN {X -91.4519,Y 23.1877,Z 96,A 159.6678,B 24.9242,C -2.0111,E1 24.8457,E2 -74.358} C_DIS
LIN {X -90.2576,Y 27.474,Z 96,A 157.7005,B 24.9218,C -2.042,E1 24.8472,E2 -72.453} C_DIS
LIN {X -89.2152,Y 30.6921,Z 96,A 155.0932,B 24.9226,C -2.0314,E1 24.8496,E2 -69.8056} C_DIS
LIN {X -87.9721,Y 34.0899,Z 96,A 153.277,B 24.9212,C -2.0498,E1 24.8513,E2 -68.0232} C_DIS
LIN {X -86.0158,Y 38.7595,Z 96,A 150.4523,B 24.9199,C -2.0669,E1 24.8544,E2 -65.2236} C_DIS
LIN {X -82.9949,Y 44.8651,Z 96,A 146.1759,B 24.9193,C -2.0748,E1 24.8598,E2 -60.9429} C_DIS
LIN {X -80.8154,Y 48.6829,Z 96,A 143.6673,B 24.9183,C -2.0874,E1 24.8633,E2 -58.4515} C_DIS
LIN {X -78.29,Y 52.6472,Z 96,A 140.615,B 24.9181,C -2.0893,E1 24.868,E2 -55.3882} C_DIS
LIN {X -76.6441,Y 55.0158,Z 96,A 138.643,B 24.9183,C -2.0872,E1 24.8712,E2 -53.4017} C_DIS
LIN {X -74.0592,Y 58.4488,Z 96,A 136.2482,B 24.9172,C -2.1009,E1 24.8752,E2 -51.028} C_DIS
LIN {X -72.0422,Y 60.9185,Z 96,A 134.0369,B 24.9175,C -2.0973,E1 24.8792,E2 -48.798} C_DIS
LIN {X -68.1346,Y 65.2594,Z 96,A 130.7291,B 24.9162,C -2.1136,E1 24.8854,E2 -45.5146} C_DIS
LIN {X -65.7287,Y 67.6822,Z 96,A 128.7274,B 24.9156,C -2.1209,E1 24.8893,E2 -43.5217} C_DIS
LIN {X -62.4789,Y 70.6946,Z 96,A 125.5292,B 24.9164,C -2.1111,E1 24.896,E2 -40.2873} C_DIS
LIN {X -58.7254,Y 73.8406,Z 96,A 123.0751,B 24.9146,C -2.134,E1 24.9012,E2 -37.8787} C_DIS
LIN {X -55.105,Y 76.5807,Z 96,A 120.0629,B 24.9148,C -2.1316,E1 24.908,E2 -34.85} C_DIS
LIN {X -52.2437,Y 78.5605,Z 96,A 117.8928,B 24.9146,C -2.1339,E1 24.9131,E2 -32.6781} C_DIS
LIN {X -48.9527,Y 80.6515,Z 96,A 115.9683,B 24.9131,C -2.1526,E1 24.9175,E2 -30.792} C_DIS
LIN {X -45.3647,Y 82.724,Z 96,A 113.3732,B 24.9129,C -2.1545,E1 24.9238,E2 -28.1937} C_DIS
LIN {X -40.4831,Y 85.2184,Z 96,A 109.5698,B 24.9137,C -2.1445,E1 24.9334,E2 -24.3565} C_DIS
LIN {X -36.4505,Y 87.0197,Z 96,A 107.0719,B 24.9129,C -2.1544,E1 24.9398,E2 -21.8761} C_DIS
LIN {X -33.2159,Y 88.305,Z 96,A 104.9417,B 24.9128,C -2.1567,E1 24.9453,E2 -19.7469} C_DIS
LIN {X -30.0622,Y 89.4276,Z 96,A 103.0943,B 24.9121,C -2.1653,E1 24.9501,E2 -17.9164} C_DIS
LIN {X -26.5431,Y 90.5349,Z 96,A 100.5656,B 24.9126,C -2.1583,E1 24.9569,E2 -15.3667} C_DIS
LIN {X -20.2081,Y 92.1557,Z 96,A 97.1404,B 24.9108,C -2.1802,E1 24.9661,E2 -11.9888} C_DIS
LIN {X -16.6849,Y 92.8582,Z 96,A 94.0631,B 24.9131,C -2.1522,E1 24.9747,E2 -8.8417} C_DIS
LIN {X -13.3506,Y 93.3959,Z 96,A 91.3929,B 24.9147,C -2.1332,E1 24.9822,E2 -6.1243} C_DIS
LIN {X -7.8095,Y 94.0219,Z 96,A 89.129,B 24.9115,C -2.172,E1 24.9883,E2 -3.9514} C_DIS
LIN {X -4.0047,Y 94.2602,Z 96,A 86.9476,B 24.9111,C -2.1774,E1 24.9943,E2 -1.7821} C_DIS
LIN {X -0.5062,Y 94.3439,Z 96,A 84.3697,B 24.9123,C -2.1627,E1 25.0016,E2 0.8309} C_DIS
LIN {X 4.0878,Y 94.2566,Z 96,A 81.8641,B 24.9115,C -2.1726,E1 25.0085,E2 3.3125} C_DIS
LIN {X 7.65,Y 94.0347,Z 96,A 79.6737,B 24.9115,C -2.1717,E1 25.0147,E2 5.5039} C_DIS
LIN {X 11.066,Y 93.694,Z 96,A 77.579,B 24.9115,C -2.1711,E1 25.0205,E2 7.5986} C_DIS
LIN {X 15.0542,Y 93.1378,Z 96,A 74.6345,B 24.913,C -2.1533,E1 25.0287,E2 10.5825} C_DIS
LIN {X 18.545,Y 92.5056,Z 96,A 72.967,B 24.9118,C -2.1691,E1 25.0332,E2 12.2107} C_DIS
LIN {X 22.9394,Y 91.5157,Z 96,A 70.1984,B 24.912,C -2.1664,E1 25.0407,E2 14.9817} C_DIS
LIN {X 25.7802,Y 90.7547,Z 96,A 68.3146,B 24.9123,C -2.1619,E1 25.0458,E2 16.8731} C_DIS
LIN {X 29.6391,Y 89.5703,Z 96,A 66.0486,B 24.912,C -2.1663,E1 25.0518,E2 19.1244} C_DIS
LIN {X 32.5276,Y 88.5608,Z 96,A 64.1338,B 24.9123,C -2.1627,E1 25.0568,E2 21.0438} C_DIS
LIN {X 39.2733,Y 85.7836,Z 96,A 59.7618,B 24.9125,C -2.16,E1 25.0681,E2 25.4119} C_DIS
LIN {X 43.0227,Y 83.9647,Z 96,A 57.2786,B 24.9126,C -2.1586,E1 25.0743,E2 27.8918} C_DIS
LIN {X 46.0863,Y 82.3231,Z 96,A 55.0904,B 24.9131,C -2.1529,E1 25.0796,E2 30.087} C_DIS
LIN {X 49.3013,Y 80.4396,Z 96,A 52.8089,B 24.9134,C -2.1489,E1 25.0851,E2 32.371} C_DIS
LIN {X 53.9415,Y 77.4038,Z 96,A 49.677,B 24.9131,C -2.1519,E1 25.0924,E2 35.4853} C_DIS
LIN {X 56.2961,Y 75.7098,Z 96,A 47.744,B 24.9139,C -2.1427,E1 25.0967,E2 37.4333} C_DIS
LIN {X 59.1658,Y 73.4883,Z 96,A 45.5836,B 24.9141,C -2.1402,E1 25.1015,E2 39.5915} C_DIS
LIN {X 61.0086,Y 71.9654,Z 96,A 43.1742,B 24.9171,C -2.1031,E1 25.1068,E2 42.0793} C_DIS
LIN {X 64.8246,Y 68.5482,Z 96,A 40.9833,B 24.9149,C -2.1298,E1 25.1111,E2 44.1982} C_DIS
LIN {X 66.8588,Y 66.5662,Z 96,A 38.7321,B 24.9167,C -2.1071,E1 25.1156,E2 46.4935} C_DIS
LIN {X 69.4551,Y 63.8515,Z 96,A 37.0717,B 24.9153,C -2.1245,E1 25.1187,E2 48.1055} C_DIS
LIN {X 71.703,Y 61.3167,Z 96,A 34.6637,B 24.9167,C -2.107,E1 25.1231,E2 50.5438} C_DIS
LIN {X 74.7012,Y 57.626,Z 96,A 31.8626,B 24.917,C -2.1033,E1 25.128,E2 53.3406} C_DIS
LIN {X 77.3879,Y 53.9644,Z 96,A 29.7446,B 24.9157,C -2.12,E1 25.1313,E2 55.409} C_DIS
LIN {X 79.0627,Y 51.482,Z 96,A 27.5706,B 24.9171,C -2.1021,E1 25.1348,E2 57.6142} C_DIS
LIN {X 80.6653,Y 48.9299,Z 96,A 25.9611,B 24.9169,C -2.1055,E1 25.1371,E2 59.2076} C_DIS
LIN {X 82.685,Y 45.4364,Z 96,A 23.2921,B 24.918,C -2.0908,E1 25.1408,E2 61.8976} C_DIS
LIN {X 84.9844,Y 40.9718,Z 96,A 20.4029,B 24.9182,C -2.0883,E1 25.1444,E2 64.7772} C_DIS
LIN {X 86.2226,Y 38.2992,Z 96,A 18.4685,B 24.919,C -2.0778,E1 25.1467,E2 66.7259} C_DIS
LIN {X 87.557,Y 35.1426,Z 96,A 16.3857,B 24.9195,C -2.0717,E1 25.1489,E2 68.8117} C_DIS
LIN {X 89.1456,Y 30.8905,Z 96,A 13.4692,B 24.9206,C -2.0577,E1 25.1517,E2 71.745} C_DIS
LIN {X 90.8681,Y 25.3798,Z 96,A 10.3709,B 24.9202,C -2.0623,E1 25.1542,E2 74.8147} C_DIS
LIN {X 92.3872,Y 19.1222,Z 96,A 6.3669,B 24.9214,C -2.0468,E1 25.1567,E2 78.8321} C_DIS
LIN {X 93.0187,Y 15.7666,Z 96,A 4.3037,B 24.9219,C -2.0407,E1 25.1578,E2 80.8977} C_DIS
LIN {X 93.5334,Y 12.352,Z 96,A 2.2307,B 24.9223,C -2.035,E1 25.1586,E2 82.9718} C_DIS
LIN {X 93.9182,Y 8.971,Z 96,A 0.143,B 24.9229,C -2.0276,E1 25.1592,E2 85.0646} C_DIS
LIN {X 94.1922,Y 5.3738,Z 96,A -2.0265,B 24.9234,C -2.0214,E1 25.1596,E2 87.2358} C_DIS
LIN {X 94.3232,Y 2.0626,Z 96,A -3.9554,B 24.9236,C -2.0181,E1 25.1598,E2 89.161} C_DIS
LIN {X 94.3398,Y -1.1605,Z 96,A -6.0744,B 24.9246,C -2.0057,E1 25.1598,E2 91.2967} C_DIS
LIN {X 94.2231,Y -4.8147,Z 96,A -7.9557,B 24.9241,C -2.0114,E1 25.1595,E2 93.1535} C_DIS
LIN {X 94.0234,Y -7.7908,Z 96,A -10.043,B 24.9254,C -1.9951,E1 25.1591,E2 95.2667} C_DIS
LIN {X 93.6574,Y -11.3787,Z 96,A -12.1773,B 24.9257,C -1.9902,E1 25.1584,E2 97.4001} C_DIS
LIN {X 93.1784,Y -14.7969,Z 96,A -14.2643,B 24.9262,C -1.9838,E1 25.1576,E2 99.4899} C_DIS
LIN {X 92.587,Y -18.1318,Z 96,A -16.0511,B 24.9259,C -1.9874,E1 25.1567,E2 101.2576} C_DIS
LIN {X 91.8842,Y -21.4092,Z 96,A -18.1157,B 24.9265,C -1.9798,E1 25.1555,E2 103.3281} C_DIS
LIN {X 90.8408,Y -25.4763,Z 96,A -20.7965,B 24.9275,C -1.9668,E1 25.1535,E2 106.0242} C_DIS
LIN {X 89.8848,Y -28.6688,Z 96,A -22.831,B 24.928,C -1.96,E1 25.1519,E2 108.0632} C_DIS
LIN {X 88.8453,Y -31.7461,Z 96,A -24.8692,B 24.9286,C -1.9514,E1 25.15,E2 110.1102} C_DIS
LIN {X 86.7603,Y -37.066,Z 96,A -28.0928,B 24.9287,C -1.9501,E1 25.1467,E2 113.3191} C_DIS
LIN {X 85.3079,Y -40.2973,Z 96,A -30.1907,B 24.929,C -1.9456,E1 25.1442,E2 115.4163} C_DIS
LIN {X 83.7145,Y -43.5102,Z 96,A -32.4933,B 24.9298,C -1.9344,E1 25.1413,E2 117.733} C_DIS
LIN {X 82.6464,Y -45.5072,Z 96,A -34.0521,B 24.9306,C -1.9235,E1 25.1392,E2 119.3094} C_DIS
LIN {X 80.5126,Y -49.1811,Z 96,A -36.5224,B 24.9309,C -1.9202,E1 25.1357,E2 121.7748} C_DIS
LIN {X 78.8591,Y -51.7908,Z 96,A -38.9035,B 24.9326,C -1.8961,E1 25.132,E2 124.2008} C_DIS
LIN {X 76.7824,Y -54.8223,Z 96,A -40.7277,B 24.932,C -1.9051,E1 25.1291,E2 125.9949} C_DIS
LIN {X 73.2194,Y -59.4976,Z 96,A -43.9053,B 24.9316,C -1.9102,E1 25.1237,E2 129.1455} C_DIS
LIN {X 70.7294,Y -62.4358,Z 96,A -46.5627,B 24.9329,C -1.8923,E1 25.1188,E2 131.8331} C_DIS
LIN {X 67.9142,Y -65.4879,Z 96,A -49.2562,B 24.9338,C -1.8796,E1 25.1136,E2 134.5448} C_DIS
LIN {X 64.2236,Y -69.1135,Z 96,A -52.2912,B 24.934,C -1.876,E1 25.1075,E2 137.5757} C_DIS
LIN {X 60.9367,Y -72.0267,Z 96,A -54.901,B 24.9343,C -1.8721,E1 25.102,E2 140.1846} C_DIS
LIN {X 56.8933,Y -75.2612,Z 96,A -57.765,B 24.9341,C -1.8756,E1 25.0957,E2 143.0297} C_DIS
LIN {X 53.215,Y -77.9059,Z 96,A -60.4426,B 24.9343,C -1.8727,E1 25.0896,E2 145.7049} C_DIS
LIN {X 50.0237,Y -79.9916,Z 96,A -62.8544,B 24.9348,C -1.8647,E1 25.0839,E2 148.1278} C_DIS
LIN {X 47.068,Y -81.7657,Z 96,A -65.449,B 24.9364,C -1.8427,E1 25.0776,E2 150.7665} C_DIS
LIN {X 44.1494,Y -83.3778,Z 96,A -67.1686,B 24.9358,C -1.8502,E1 25.0734,E2 152.4633} C_DIS
LIN {X 40.5275,Y -85.1977,Z 96,A -69.6424,B 24.9361,C -1.8458,E1 25.0672,E2 154.9411} C_DIS
LIN {X 36.7653,Y -86.887,Z 96,A -72.2111,B 24.9366,C -1.8398,E1 25.0606,E2 157.5179} C_DIS
LIN {X 30.8073,Y -89.1748,Z 96,A -75.8334,B 24.9363,C -1.8437,E1 25.0511,E2 161.1232} C_DIS
LIN {X 27.676,Y -90.195,Z 96,A -77.8787,B 24.9366,C -1.8397,E1 25.0457,E2 163.1743} C_DIS
LIN {X 24.8223,Y -91.0216,Z 96,A -79.9727,B 24.9374,C -1.8275,E1 25.04,E2 165.2939} C_DIS
LIN {X 17.2318,Y -92.7598,Z 96,A -84.3766,B 24.9369,C -1.8347,E1 25.028,E2 169.6749} C_DIS
LIN {X 13.8731,Y -93.3206,Z 96,A -86.402,B 24.9369,C -1.8347,E1 25.0224,E2 171.6983} C_DIS
LIN {X 10.6983,Y -93.7371,Z 96,A -88.3998,B 24.9371,C -1.8316,E1 25.0169,E2 173.7019} C_DIS
LIN {X 7.1903,Y -94.0714,Z 96,A -90.5122,B 24.9371,C -1.8315,E1 25.011,E2 175.8134} C_DIS
LIN {X 3.8518,Y -94.2668,Z 96,A -92.5551,B 24.9372,C -1.8303,E1 25.0053,E2 177.8584} C_DIS
LIN {X 0.6541,Y -94.3407,Z 96,A -93.7059,B 24.9353,C -1.8575,E1 25.0023,E2 178.9445} C_DIS
Enddeposition()
LIN {X 0.6541,Y -94.3407,Z 96,A -93.7059,B 24.9353,C -1.8575,E1 25.0023,E2 178.9445} C_DIS
Startdeposition()
$VEL.CP = VEL_PRINT
LIN {X 1.3977,Y -93.4214,Z 96,A -93.1094,B 24.9339,C -1.8783,E1 25.0041,E2 178.2988} C_DIS
LIN {X 4.5839,Y -93.3205,Z 96,A -91.0032,B 24.9334,C -1.8843,E1 25.01,E2 176.179} C_DIS
LIN {X 8.0452,Y -93.0859,Z 96,A -88.9061,B 24.9334,C -1.8843,E1 25.0158,E2 174.083} C_DIS
LIN {X 11.1031,Y -92.7695,Z 96,A -87.0713,B 24.9334,C -1.8836,E1 25.0209,E2 172.2511} C_DIS
LIN {X 15.5148,Y -92.1342,Z 96,A -84.5008,B 24.9338,C -1.8798,E1 25.028,E2 169.692} C_DIS
LIN {X 19.4106,Y -91.3939,Z 96,A -81.604,B 24.9324,C -1.8985,E1 25.036,E2 166.7545} C_DIS
LIN {X 24.0044,Y -90.2958,Z 96,A -79.0255,B 24.933,C -1.89,E1 25.0429,E2 164.2} C_DIS
LIN {X 27.2329,Y -89.3755,Z 96,A -76.984,B 24.933,C -1.8917,E1 25.0484,E2 162.158} C_DIS
LIN {X 30.4898,Y -88.3176,Z 96,A -74.8979,B 24.9328,C -1.8938,E1 25.0539,E2 160.071} C_DIS
LIN {X 34.4604,Y -86.8446,Z 96,A -72.333,B 24.9326,C -1.8962,E1 25.0606,E2 157.506} C_DIS
LIN {X 37.3367,Y -85.6468,Z 96,A -70.5163,B 24.9326,C -1.8956,E1 25.0652,E2 155.695} C_DIS
LIN {X 41.4914,Y -83.713,Z 96,A -66.5776,B 24.9293,C -1.9416,E1 25.0754,E2 151.6579} C_DIS
LIN {X 46.2745,Y -81.1676,Z 96,A -64.6108,B 24.9325,C -1.8974,E1 25.0799,E2 149.8012} C_DIS
LIN {X 48.3793,Y -79.9305,Z 96,A -62.857,B 24.9316,C -1.9096,E1 25.0842,E2 148.0242} C_DIS
LIN {X 51.0374,Y -78.2612,Z 96,A -60.796,B 24.931,C -1.9183,E1 25.089,E2 145.9493} C_DIS
LIN {X 55.7242,Y -74.9964,Z 96,A -57.3734,B 24.9307,C -1.9225,E1 25.0968,E2 142.5287} C_DIS
LIN {X 58.5069,Y -72.8458,Z 96,A -55.0136,B 24.9298,C -1.9347,E1 25.102,E2 140.1488} C_DIS
LIN {X 62.3944,Y -69.5439,Z 96,A -51.8888,B 24.9293,C -1.9418,E1 25.1086,E2 137.0196} C_DIS
LIN {X 64.6919,Y -67.4122,Z 96,A -49.83,B 24.9286,C -1.9515,E1 25.1128,E2 134.9464} C_DIS
LIN {X 66.9643,Y -65.1563,Z 96,A -48.0415,B 24.9287,C -1.9497,E1 25.1163,E2 133.1697} C_DIS
LIN {X 70.1452,Y -61.7176,Z 96,A -45.0684,B 24.9279,C -1.9608,E1 25.1218,E2 130.1837} C_DIS
LIN {X 73.548,Y -57.6216,Z 96,A -41.2495,B 24.9257,C -1.9904,E1 25.1286,E2 126.3127} C_DIS
LIN {X 76.5346,Y -53.5907,Z 96,A -39.0912,B 24.9277,C -1.9641,E1 25.1319,E2 124.2271} C_DIS
LIN {X 78.0354,Y -51.3798,Z 96,A -37.5665,B 24.9277,C -1.9644,E1 25.1343,E2 122.7093} C_DIS
LIN {X 79.8001,Y -48.5938,Z 96,A -35.5362,B 24.9272,C -1.9704,E1 25.1373,E2 120.675} C_DIS
LIN {X 81.9793,Y -44.8206,Z 96,A -31.8259,B 24.9237,C -2.0177,E1 25.1424,E2 116.8724} C_DIS
LIN {X 84.3867,Y -40.1055,Z 96,A -29.9447,B 24.9268,C -1.9755,E1 25.1446,E2 115.1011} C_DIS
LIN {X 85.769,Y -37.0565,Z 96,A -27.3944,B 24.925,C -2.0005,E1 25.1475,E2 112.5056} C_DIS
LIN {X 87.264,Y -33.384,Z 96,A -25.1566,B 24.925,C -2.0006,E1 25.1498,E2 110.2799} C_DIS
LIN {X 88.2788,Y -30.6004,Z 96,A -23.3442,B 24.9245,C -2.0061,E1 25.1515,E2 108.4648} C_DIS
LIN {X 89.2798,Y -27.5416,Z 96,A -21.3956,B 24.9241,C -2.0113,E1 25.1531,E2 106.5149} C_DIS
LIN {X 90.2879,Y -24.0337,Z 96,A -18.9462,B 24.923,C -2.0264,E1 25.155,E2 104.044} C_DIS
LIN {X 91.3376,Y -19.67,Z 96,A -16.6027,B 24.9235,C -2.0196,E1 25.1564,E2 101.7301} C_DIS
LIN {X 91.9142,Y -16.77,Z 96,A -14.6017,B 24.9225,C -2.0325,E1 25.1575,E2 99.7102} C_DIS
LIN {X 92.5234,Y -12.9941,Z 96,A -12.4152,B 24.9225,C -2.034,E1 25.1584,E2 97.5331} C_DIS
LIN {X 92.8851,Y -10.0948,Z 96,A -10.5082,B 24.9216,C -2.0442,E1 25.159,E2 95.6135} C_DIS
LIN {X 93.2029,Y -6.5332,Z 96,A -8.3491,B 24.9212,C -2.05,E1 25.1595,E2 93.4535} C_DIS
LIN {X 93.3837,Y -2.9854,Z 96,A -6.2392,B 24.9209,C -2.0544,E1 25.1597,E2 91.3457} C_DIS
LIN {X 93.4331,Y 0.015,Z 96,A -4.2624,B 24.92,C -2.0654,E1 25.1597,E2 89.3545} C_DIS
LIN {X 93.3636,Y 3.5813,Z 96,A -2.149,B 24.9197,C -2.0697,E1 25.1596,E2 87.2438} C_DIS
LIN {X 93.1558,Y 7.1748,Z 96,A -0.0079,B 24.9193,C -2.0742,E1 25.1592,E2 85.1047} C_DIS
LIN {X 92.8242,Y 10.6361,Z 96,A 2.0824,B 24.9189,C -2.0794,E1 25.1586,E2 83.0145} C_DIS
LIN {X 92.3782,Y 13.9914,Z 96,A 4.1683,B 24.9184,C -2.0863,E1 25.1578,E2 80.9246} C_DIS
LIN {X 91.8032,Y 17.3687,Z 96,A 6.2445,B 24.9179,C -2.0919,E1 25.1567,E2 78.8472} C_DIS
LIN {X 90.895,Y 21.628,Z 96,A 8.7464,B 24.9178,C -2.0938,E1 25.1552,E2 76.3555} C_DIS
LIN {X 89.9804,Y 25.1602,Z 96,A 11.1174,B 24.9168,C -2.1057,E1 25.1535,E2 73.9701} C_DIS
LIN {X 89.0658,Y 28.2312,Z 96,A 13.5584,B 24.9149,C -2.1295,E1 25.1515,E2 71.4867} C_DIS
LIN {X 88.0226,Y 31.3306,Z 96,A 14.9482,B 24.9163,C -2.1123,E1 25.1502,E2 70.1454} C_DIS
LIN {X 87.2763,Y 33.3516,Z 96,A 16.2762,B 24.916,C -2.1164,E1 25.1489,E2 68.8151} C_DIS
LIN {X 86.1133,Y 36.2479,Z 96,A 18.2982,B 24.9152,C -2.126,E1 25.1467,E2 66.7816} C_DIS
LIN {X 84.4882,Y 39.8924,Z 96,A 20.8533,B 24.9144,C -2.137,E1 25.1438,E2 64.2144} C_DIS
LIN {X 81.3236,Y 46.0016,Z 96,A 24.9361,B 24.9138,C -2.1434,E1 25.1384,E2 60.138} C_DIS
LIN {X 80.0854,Y 48.1244,Z 96,A 26.4968,B 24.9134,C -2.1494,E1 25.1362,E2 58.5712} C_DIS
LIN {X 78.1654,Y 51.1826,Z 96,A 28.5718,B 24.9134,C -2.1499,E1 25.1331,E2 56.5052} C_DIS
LIN {X 76.3967,Y 53.7891,Z 96,A 30.6242,B 24.9126,C -2.1593,E1 25.1298,E2 54.4408} C_DIS
LIN {X 74.2183,Y 56.7553,Z 96,A 32.7641,B 24.9125,C -2.1605,E1 25.1262,E2 52.3083} C_DIS
LIN {X 72.356,Y 59.1114,Z 96,A 34.785,B 24.9116,C -2.1715,E1 25.1226,E2 50.2709} C_DIS
LIN {X 69.7029,Y 62.2168,Z 96,A 37.1021,B 24.9116,C -2.1703,E1 25.1184,E2 47.967} C_DIS
LIN {X 67.01,Y 65.1092,Z 96,A 39.3519,B 24.9117,C -2.1692,E1 25.1141,E2 45.7295} C_DIS
LIN {X 65.0884,Y 67.03,Z 96,A 41.2059,B 24.9109,C -2.1796,E1 25.1104,E2 43.8587} C_DIS
LIN {X 62.5026,Y 69.447,Z 96,A 43.7017,B 24.9096,C -2.1959,E1 25.1052,E2 41.3345} C_DIS
LIN {X 58.957,Y 72.4811,Z 96,A 46.1567,B 24.9103,C -2.1865,E1 25.1,E2 38.9112} C_DIS
LIN {X 56.8071,Y 74.1784,Z 96,A 47.9192,B 24.9098,C -2.1925,E1 25.0961,E2 37.1409} C_DIS
LIN {X 54.0851,Y 76.1857,Z 96,A 49.8117,B 24.9101,C -2.1896,E1 25.0918,E2 35.262} C_DIS
LIN {X 51.1513,Y 78.1861,Z 96,A 52.1835,B 24.9092,C -2.2001,E1 25.0863,E2 32.8733} C_DIS
LIN {X 47.9776,Y 80.1736,Z 96,A 54.4922,B 24.9089,C -2.204,E1 25.0808,E2 30.5627} C_DIS
LIN {X 44.7195,Y 82.0342,Z 96,A 56.7127,B 24.9089,C -2.2043,E1 25.0754,E2 28.3478} C_DIS
LIN {X 41.8116,Y 83.5543,Z 96,A 58.818,B 24.9084,C -2.2102,E1 25.0701,E2 26.2344} C_DIS
LIN {X 38.3337,Y 85.2053,Z 96,A 61.7405,B 24.9065,C -2.233,E1 25.0626,E2 23.2652} C_DIS
LIN {X 34.5352,Y 86.8153,Z 96,A 63.3373,B 24.909,C -2.2024,E1 25.0587,E2 21.7445} C_DIS
LIN {X 31.8502,Y 87.8351,Z 96,A 65.2442,B 24.9085,C -2.2092,E1 25.0536,E2 19.8256} C_DIS
LIN {X 28.6433,Y 88.9325,Z 96,A 67.3264,B 24.9083,C -2.211,E1 25.0481,E2 17.743} C_DIS
LIN {X 25.6258,Y 89.8485,Z 96,A 69.3263,B 24.908,C -2.2147,E1 25.0427,E2 15.7378} C_DIS
LIN {X 22.4153,Y 90.703,Z 96,A 71.374,B 24.9079,C -2.2163,E1 25.0372,E2 13.6895} C_DIS
LIN {X 18.6987,Y 91.5411,Z 96,A 73.6438,B 24.9079,C -2.2152,E1 25.031,E2 11.4254} C_DIS
LIN {X 14.0746,Y 92.3653,Z 96,A 76.4754,B 24.908,C -2.2145,E1 25.0232,E2 8.5984} C_DIS
LIN {X 10.8538,Y 92.7987,Z 96,A 78.526,B 24.9078,C -2.2169,E1 25.0175,E2 6.5437} C_DIS
LIN {X 7.331,Y 93.1433,Z 96,A 80.7941,B 24.9075,C -2.2204,E1 25.0112,E2 4.2685} C_DIS
LIN {X 3.9276,Y 93.3487,Z 96,A 82.8691,B 24.9075,C -2.2198,E1 25.0054,E2 2.1957} C_DIS
LIN {X -1.8654,Y 93.4128,Z 96,A 86.1628,B 24.9084,C -2.2103,E1 24.9963,E2 -1.0753} C_DIS
LIN {X -6.0667,Y 93.2344,Z 96,A 88.6413,B 24.9087,C -2.206,E1 24.9894,E2 -3.5442} C_DIS
LIN {X -13.6506,Y 92.4301,Z 96,A 93.5149,B 24.9084,C -2.2099,E1 24.9759,E2 -8.4301} C_DIS
LIN {X -19.3387,Y 91.4097,Z 96,A 97.2456,B 24.9081,C -2.2133,E1 24.9656,E2 -12.173} C_DIS
LIN {X -22.4802,Y 90.6872,Z 96,A 99.2433,B 24.9081,C -2.2122,E1 24.9602,E2 -14.1707} C_DIS
LIN {X -27.4565,Y 89.3062,Z 96,A 102.2682,B 24.9089,C -2.2041,E1 24.9521,E2 -17.1812} C_DIS
LIN {X -30.0781,Y 88.4577,Z 96,A 104.1284,B 24.9086,C -2.2077,E1 24.9471,E2 -19.0533} C_DIS
LIN {X -33.5812,Y 87.1894,Z 96,A 106.4483,B 24.9087,C -2.2058,E1 24.9411,E2 -21.3737} C_DIS
LIN {X -37.6854,Y 85.4948,Z 96,A 108.9255,B 24.9097,C -2.1939,E1 24.9347,E2 -23.8282} C_DIS
LIN {X -41.7703,Y 83.5748,Z 96,A 112.3854,B 24.9082,C -2.2121,E1 24.9259,E2 -27.3404} C_DIS
LIN {X -44.873,Y 81.951,Z 96,A 113.8837,B 24.9103,C -2.1874,E1 24.9224,E2 -28.7839} C_DIS
LIN {X -47.6498,Y 80.3674,Z 96,A 116.0485,B 24.91,C -2.1905,E1 24.9171,E2 -30.9627} C_DIS
LIN {X -50.8746,Y 78.3672,Z 96,A 118.4524,B 24.9102,C -2.1886,E1 24.9114,E2 -33.3697} C_DIS
LIN {X -53.1286,Y 76.8558,Z 96,A 120.9387,B 24.9082,C -2.2119,E1 24.9056,E2 -35.92} C_DIS
LIN {X -57.1312,Y 73.9287,Z 96,A 122.8228,B 24.9118,C -2.1682,E1 24.9016,E2 -37.7069} C_DIS
LIN {X -59.014,Y 72.4349,Z 96,A 124.5995,B 24.9113,C -2.1747,E1 24.8977,E2 -39.5056} C_DIS
LIN {X -61.9718,Y 69.9222,Z 96,A 126.9985,B 24.9117,C -2.1699,E1 24.8927,E2 -41.9026} C_DIS
LIN {X -64.6782,Y 67.4254,Z 96,A 129.1638,B 24.9124,C -2.1617,E1 24.8883,E2 -44.0572} C_DIS
LIN {X -67.137,Y 64.9774,Z 96,A 131.3335,B 24.9127,C -2.1579,E1 24.884,E2 -46.227} C_DIS
LIN {X -69.7683,Y 62.1437,Z 96,A 133.6136,B 24.9134,C -2.149,E1 24.8797,E2 -48.4962} C_DIS
LIN {X -71.8656,Y 59.7054,Z 96,A 135.6943,B 24.9135,C -2.1474,E1 24.876,E2 -50.5825} C_DIS
LIN {X -73.9691,Y 57.0787,Z 96,A 137.7308,B 24.914,C -2.1411,E1 24.8725,E2 -52.6135} C_DIS
LIN {X -76.3858,Y 53.8045,Z 96,A 140.2624,B 24.9145,C -2.1354,E1 24.8683,E2 -55.1439} C_DIS
LIN {X -79.5031,Y 49.0806,Z 96,A 143.7437,B 24.9152,C -2.126,E1 24.8631,E2 -58.6202} C_DIS
LIN {X -81.2677,Y 46.1003,Z 96,A 146.0222,B 24.9153,C -2.1247,E1 24.8599,E2 -60.9076} C_DIS
LIN {X -83.5133,Y 41.8944,Z 96,A 148.6429,B 24.9168,C -2.1067,E1 24.8565,E2 -63.4992} C_DIS
LIN {X -85.201,Y 38.3431,Z 96,A 151.2921,B 24.9168,C -2.1069,E1 24.8534,E2 -66.1634} C_DIS
LIN {X -86.572,Y 35.1384,Z 96,A 153.8086,B 24.9163,C -2.1122,E1 24.8506,E2 -68.7066} C_DIS
LIN {X -88.3165,Y 30.493,Z 96,A 156.5555,B 24.9178,C -2.0935,E1 24.8481,E2 -71.4244} C_DIS
LIN {X -89.4257,Y 27.0688,Z 96,A 159.0587,B 24.9176,C -2.0959,E1 24.846,E2 -73.9476} C_DIS
LIN {X -90.3732,Y 23.7132,Z 96,A 160.9348,B 24.9188,C -2.0809,E1 24.8446,E2 -75.799} C_DIS
LIN {X -91.1922,Y 20.3365,Z 96,A 163.1284,B 24.9192,C -2.0761,E1 24.8433,E2 -77.9941} C_DIS
LIN {X -92.0636,Y 15.9368,Z 96,A 165.6296,B 24.9205,C -2.0596,E1 24.842,E2 -80.4706} C_DIS
LIN {X -92.8428,Y 10.4773,Z 96,A 169.2821,B 24.9206,C -2.0572,E1 24.8406,E2 -84.1391} C_DIS
LIN {X -93.1736,Y 6.9511,Z 96,A 171.4505,B 24.9212,C -2.0501,E1 24.8401,E2 -86.3035} C_DIS
LIN {X -93.3784,Y 3.1572,Z 96,A 174.274,B 24.9206,C -2.058,E1 24.8398,E2 -89.1629} C_DIS
LIN {X -93.4312,Y -0.3935,Z 96,A 175.5906,B 24.9232,C -2.0242,E1 24.8398,E2 -90.4069} C_DIS
LIN {X -93.39,Y -2.7779,Z 96,A 178.0795,B 24.9211,C -2.0515,E1 24.84,E2 -92.976} C_DIS
LIN {X -93.18,Y -6.8686,Z 96,A -179.2618,B 24.9213,C -2.0481,E1 24.8406,E2 -95.6425} C_DIS
LIN {X -92.746,Y -11.3039,Z 96,A -177.4604,B 24.9242,C -2.0103,E1 24.8411,E2 -97.3644} C_DIS
LIN {X -91.8319,Y -17.2196,Z 96,A -173.6224,B 24.9247,C -2.004,E1 24.8428,E2 -101.2101} C_DIS
LIN {X -91.1279,Y -20.6222,Z 96,A -171.4087,B 24.925,C -2,E1 24.8441,E2 -103.4273} C_DIS
LIN {X -90.3878,Y -23.6562,Z 96,A -169.4711,B 24.9254,C -1.9948,E1 24.8455,E2 -105.3639} C_DIS
LIN {X -89.4027,Y -27.1451,Z 96,A -167.3109,B 24.926,C -1.9861,E1 24.8472,E2 -107.5159} C_DIS
LIN {X -88.5788,Y -29.719,Z 96,A -165.6213,B 24.9263,C -1.9822,E1 24.8486,E2 -109.2058} C_DIS
LIN {X -87.3558,Y -33.1417,Z 96,A -163.1836,B 24.9263,C -1.9822,E1 24.851,E2 -111.6574} C_DIS
LIN {X -85.8101,Y -36.9621,Z 96,A -160.7795,B 24.9272,C -1.9711,E1 24.8536,E2 -114.0482} C_DIS
LIN {X -84.2677,Y -40.3531,Z 96,A -158.575,B 24.9278,C -1.9621,E1 24.8562,E2 -116.2434} C_DIS
LIN {X -82.0331,Y -44.7215,Z 96,A -155.6878,B 24.9287,C -1.95,E1 24.8599,E2 -119.117} C_DIS
LIN {X -80.7282,Y -47.0391,Z 96,A -153.7775,B 24.9284,C -1.9545,E1 24.8626,E2 -121.048} C_DIS
LIN {X -78.9673,Y -49.9383,Z 96,A -151.6806,B 24.9287,C -1.9496,E1 24.8657,E2 -123.1439} C_DIS
LIN {X -77.2736,Y -52.5188,Z 96,A -148.7308,B 24.9266,C -1.979,E1 24.8705,E2 -126.1783} C_DIS
LIN {X -73.9152,Y -57.1486,Z 96,A -146.9198,B 24.9312,C -1.9157,E1 24.8733,E2 -127.8473} C_DIS
LIN {X -71.6038,Y -60.0205,Z 96,A -143.9536,B 24.93,C -1.933,E1 24.8786,E2 -130.8684} C_DIS
LIN {X -69.2773,Y -62.6922,Z 96,A -141.8222,B 24.9304,C -1.9267,E1 24.8825,E2 -132.9945} C_DIS
LIN {X -66.8363,Y -65.2884,Z 96,A -139.6408,B 24.9308,C -1.9219,E1 24.8867,E2 -135.1737} C_DIS
LIN {X -64.3722,Y -67.7191,Z 96,A -137.4492,B 24.9309,C -1.9197,E1 24.8912,E2 -137.3693} C_DIS
LIN {X -61.5255,Y -70.3137,Z 96,A -135.2366,B 24.9316,C -1.9102,E1 24.8957,E2 -139.5681} C_DIS
LIN {X -58.9015,Y -72.5261,Z 96,A -133.0988,B 24.9318,C -1.9074,E1 24.9003,E2 -141.7073} C_DIS
LIN {X -56.0363,Y -74.762,Z 96,A -130.9493,B 24.9323,C -1.9008,E1 24.9051,E2 -143.8489} C_DIS
LIN {X -51.1756,Y -78.1701,Z 96,A -127.3194,B 24.9327,C -1.8945,E1 24.9134,E2 -147.476} C_DIS
LIN {X -48.3848,Y -79.9271,Z 96,A -125.0996,B 24.9325,C -1.898,E1 24.9187,E2 -149.7111} C_DIS
LIN {X -45.0865,Y -81.8344,Z 96,A -122.6653,B 24.9325,C -1.898,E1 24.9247,E2 -152.1525} C_DIS
LIN {X -41.9966,Y -83.4626,Z 96,A -120.5807,B 24.9328,C -1.8934,E1 24.9298,E2 -154.2318} C_DIS
LIN {X -37.2717,Y -85.6752,Z 96,A -117.6254,B 24.9336,C -1.8816,E1 24.9373,E2 -157.1664} C_DIS
LIN {X -34.4946,Y -86.8312,Z 96,A -115.6733,B 24.9336,C -1.8833,E1 24.9424,E2 -159.1269} C_DIS
LIN {X -31.7912,Y -87.8566,Z 96,A -113.8804,B 24.9336,C -1.8824,E1 24.9471,E2 -160.9214} C_DIS
LIN {X -28.9477,Y -88.834,Z 96,A -111.9859,B 24.9336,C -1.8827,E1 24.9521,E2 -162.82} C_DIS
LIN {X -25.6665,Y -89.8369,Z 96,A -109.9094,B 24.9337,C -1.8803,E1 24.9576,E2 -164.8943} C_DIS
LIN {X -22.0821,Y -90.7843,Z 96,A -107.8836,B 24.9344,C -1.8705,E1 24.9631,E2 -166.8998} C_DIS
LIN {X -17.6318,Y -91.7525,Z 96,A -104.8676,B 24.934,C -1.8769,E1 24.9714,E2 -169.9345} C_DIS
LIN {X -14.0391,Y -92.3708,Z 96,A -102.6861,B 24.9341,C -1.8744,E1 24.9774,E2 -172.1122} C_DIS
LIN {X -10.6502,Y -92.8225,Z 96,A -100.4346,B 24.9338,C -1.8794,E1 24.9836,E2 -174.3771} C_DIS
LIN {X -7.2013,Y -93.1537,Z 96,A -98.3057,B 24.9338,C -1.8794,E1 24.9896,E2 -176.5071} C_DIS
LIN {X -3.439,Y -93.3697,Z 96,A -96.0298,B 24.9338,C -1.8783,E1 24.9959,E2 -178.781} C_DIS
LIN {X -0.4343,Y -93.4304,Z 96,A -94.1693,B 24.9338,C -1.8793,E1 25.0011,E2 -180.6439} C_DIS
LIN {X -0.4343,Y -93.4304,Z 96,A -94.1693,B 24.9338,C -1.8793,E1 25.0011,E2 -180.6439} C_DIS
Enddeposition()
LIN {X 0.6474,Y -92.5151,Z 96,A -94.4167,B 24.9349,C -1.864,E1 25.0003,E2 -180.3601} C_DIS
Startdeposition()
$VEL.CP = VEL_PRINT
LIN {X -2.2714,Y -92.4912,Z 96,A -96.175,B 24.9348,C -1.8653,E1 24.9954,E2 -178.6048} C_DIS
LIN {X -4.5371,Y -92.4078,Z 96,A -97.7794,B 24.9353,C -1.8584,E1 24.9909,E2 -176.9836} C_DIS
LIN {X -7.9455,Y -92.1772,Z 96,A -99.8871,B 24.9353,C -1.8587,E1 24.985,E2 -174.8758} C_DIS
LIN {X -10.8494,Y -91.879,Z 96,A -101.503,B 24.9348,C -1.8654,E1 24.9806,E2 -173.2748} C_DIS
LIN {X -13.5735,Y -91.518,Z 96,A -103.2061,B 24.9348,C -1.8657,E1 24.9759,E2 -171.571} C_DIS
LIN {X -16.3723,Y -91.0572,Z 96,A -105.0911,B 24.935,C -1.8619,E1 24.9706,E2 -169.6754} C_DIS
LIN {X -19.8179,Y -90.3699,Z 96,A -107.2211,B 24.9348,C -1.8644,E1 24.9648,E2 -167.5487} C_DIS
LIN {X -22.4955,Y -89.7425,Z 96,A -109.0372,B 24.935,C -1.8615,E1 24.9599,E2 -165.7233} C_DIS
LIN {X -25.3108,Y -88.9878,Z 96,A -110.6539,B 24.9345,C -1.8689,E1 24.9556,E2 -164.1217} C_DIS
LIN {X -27.9392,Y -88.1996,Z 96,A -112.3568,B 24.9345,C -1.87,E1 24.951,E2 -162.4184} C_DIS
LIN {X -30.1083,Y -87.4829,Z 96,A -113.7729,B 24.9344,C -1.8711,E1 24.9473,E2 -161.0022} C_DIS
LIN {X -32.2423,Y -86.7191,Z 96,A -115.3811,B 24.9348,C -1.8657,E1 24.943,E2 -159.3777} C_DIS
LIN {X -35.4068,Y -85.4759,Z 96,A -117.5055,B 24.9346,C -1.8671,E1 24.9375,E2 -157.2522} C_DIS
LIN {X -38.5481,Y -84.1059,Z 96,A -119.6061,B 24.9344,C -1.8702,E1 24.9322,E2 -155.1537} C_DIS
LIN {X -41.1704,Y -82.8521,Z 96,A -121.2215,B 24.9339,C -1.8784,E1 24.9281,E2 -153.5536} C_DIS
LIN {X -43.6037,Y -81.5996,Z 96,A -123.1208,B 24.9342,C -1.8739,E1 24.9234,E2 -151.6385} C_DIS
LIN {X -46.1754,Y -80.1704,Z 96,A -124.8332,B 24.9337,C -1.88,E1 24.9193,E2 -149.9356} C_DIS
LIN {X -48.5253,Y -78.7723,Z 96,A -126.4496,B 24.9334,C -1.8849,E1 24.9154,E2 -148.3259} C_DIS
LIN {X -50.4517,Y -77.5526,Z 96,A -128.1327,B 24.9339,C -1.8784,E1 24.9114,E2 -146.6218} C_DIS
LIN {X -53.1053,Y -75.7589,Z 96,A -129.9178,B 24.9332,C -1.888,E1 24.9074,E2 -144.8535} C_DIS
LIN {X -55.6004,Y -73.9463,Z 96,A -131.8728,B 24.933,C -1.8899,E1 24.903,E2 -142.8961} C_DIS
LIN {X -58.2531,Y -71.8751,Z 96,A -133.975,B 24.9328,C -1.8931,E1 24.8984,E2 -140.7937} C_DIS
LIN {X -60.8589,Y -69.6825,Z 96,A -136.1026,B 24.9326,C -1.8965,E1 24.8938,E2 -138.6661} C_DIS
LIN {X -63.387,Y -67.391,Z 96,A -138.2184,B 24.9323,C -1.9007,E1 24.8895,E2 -136.5516} C_DIS
LIN {X -65.8219,Y -65.0149,Z 96,A -140.3323,B 24.932,C -1.9049,E1 24.8853,E2 -134.4389} C_DIS
LIN {X -68.1655,Y -62.5534,Z 96,A -142.4486,B 24.9317,C -1.9092,E1 24.8813,E2 -132.3233} C_DIS
LIN {X -70.4168,Y -60.0078,Z 96,A -144.5155,B 24.9312,C -1.9151,E1 24.8775,E2 -130.2613} C_DIS
LIN {X -72.421,Y -57.5737,Z 96,A -146.5483,B 24.9311,C -1.9172,E1 24.8739,E2 -128.224} C_DIS
LIN {X -74.3712,Y -55.0327,Z 96,A -148.6198,B 24.9309,C -1.9193,E1 24.8704,E2 -126.1476} C_DIS
LIN {X -76.0737,Y -52.6525,Z 96,A -150.2723,B 24.9303,C -1.9288,E1 24.8678,E2 -124.5096} C_DIS
LIN {X -77.8158,Y -50.0416,Z 96,A -152.2374,B 24.9299,C -1.9331,E1 24.8648,E2 -122.5449} C_DIS
LIN {X -79.3573,Y -47.5626,Z 96,A -154.2016,B 24.9299,C -1.933,E1 24.8619,E2 -120.5704} C_DIS
LIN {X -80.8167,Y -45.0347,Z 96,A -155.8257,B 24.9292,C -1.9435,E1 24.8597,E2 -118.963} C_DIS
LIN {X -82.1335,Y -42.5893,Z 96,A -157.7458,B 24.9292,C -1.942,E1 24.8572,E2 -117.029} C_DIS
LIN {X -83.4316,Y -39.983,Z 96,A -159.4523,B 24.9287,C -1.9501,E1 24.8551,E2 -115.3324} C_DIS
LIN {X -84.5811,Y -37.4941,Z 96,A -161.0791,B 24.9282,C -1.957,E1 24.8532,E2 -113.7134} C_DIS
LIN {X -85.6533,Y -34.9711,Z 96,A -162.9272,B 24.9282,C -1.9573,E1 24.8512,E2 -111.8557} C_DIS
LIN {X -86.8868,Y -31.7829,Z 96,A -164.9676,B 24.9275,C -1.9658,E1 24.8492,E2 -109.8242} C_DIS
LIN {X -87.6942,Y -29.4819,Z 96,A -166.4386,B 24.9271,C -1.9715,E1 24.8479,E2 -108.3583} C_DIS
LIN {X -88.5379,Y -26.8479,Z 96,A -168.2736,B 24.9271,C -1.9729,E1 24.8463,E2 -106.5161} C_DIS
LIN {X -89.3388,Y -24.0425,Z 96,A -169.9813,B 24.9264,C -1.9814,E1 24.8451,E2 -104.8188} C_DIS
LIN {X -90.0147,Y -21.3805,Z 96,A -171.6946,B 24.926,C -1.9862,E1 24.8439,E2 -103.107} C_DIS
LIN {X -90.611,Y -18.6845,Z 96,A -173.5078,B 24.9259,C -1.9884,E1 24.8429,E2 -101.2883} C_DIS
LIN {X -91.1636,Y -15.7775,Z 96,A -175.4885,B 24.9258,C -1.9896,E1 24.8419,E2 -99.2988} C_DIS
LIN {X -91.6714,Y -12.4935,Z 96,A -177.5303,B 24.9253,C -1.9966,E1 24.8411,E2 -97.2613} C_DIS
LIN {X -92.0337,Y -9.449,Z 96,A -179.3357,B 24.9246,C -2.0054,E1 24.8405,E2 -95.4663} C_DIS
LIN {X -92.3041,Y -6.2785,Z 96,A 178.6336,B 24.9243,C -2.0099,E1 24.8401,E2 -93.434} C_DIS
LIN {X -92.4768,Y -2.7396,Z 96,A 176.5621,B 24.9234,C -2.0206,E1 24.8398,E2 -91.3755} C_DIS
LIN {X -92.5187,Y -0.1097,Z 96,A 174.9047,B 24.9231,C -2.0249,E1 24.8398,E2 -89.7185} C_DIS
LIN {X -92.4918,Y 2.241,Z 96,A 173.4394,B 24.9228,C -2.0293,E1 24.8398,E2 -88.2549} C_DIS
LIN {X -92.3802,Y 5.037,Z 96,A 171.6608,B 24.9225,C -2.0335,E1 24.8401,E2 -86.4756} C_DIS
LIN {X -92.1776,Y 7.9415,Z 96,A 169.6988,B 24.9224,C -2.0345,E1 24.8405,E2 -84.5041} C_DIS
LIN {X -91.8803,Y 10.8384,Z 96,A 168.0767,B 24.9215,C -2.0458,E1 24.841,E2 -82.8992} C_DIS
LIN {X -91.5169,Y 13.5807,Z 96,A 166.3527,B 24.9211,C -2.0509,E1 24.8417,E2 -81.1772} C_DIS
LIN {X -91.0727,Y 16.286,Z 96,A 164.5859,B 24.9209,C -2.0543,E1 24.8425,E2 -79.408} C_DIS
LIN {X -90.6084,Y 18.6971,Z 96,A 163.1097,B 24.9204,C -2.0605,E1 24.8433,E2 -77.9378} C_DIS
LIN {X -90.0159,Y 21.3756,Z 96,A 161.3979,B 24.92,C -2.0654,E1 24.8444,E2 -76.2278} C_DIS
LIN {X -89.341,Y 24.0344,Z 96,A 159.638,B 24.9197,C -2.069,E1 24.8456,E2 -74.4661} C_DIS
LIN {X -88.671,Y 26.3993,Z 96,A 158.0717,B 24.9195,C -2.0724,E1 24.8468,E2 -72.899} C_DIS
LIN {X -87.8495,Y 29.0216,Z 96,A 156.4409,B 24.9189,C -2.0798,E1 24.8482,E2 -71.2765} C_DIS
LIN {X -87.0954,Y 31.2109,Z 96,A 154.7694,B 24.9191,C -2.0771,E1 24.8498,E2 -69.589} C_DIS
LIN {X -85.8959,Y 34.3753,Z 96,A 152.6978,B 24.9185,C -2.0843,E1 24.8519,E2 -67.5228} C_DIS
LIN {X -84.7712,Y 37.0582,Z 96,A 151.0746,B 24.9177,C -2.0951,E1 24.8536,E2 -65.9166} C_DIS
LIN {X -83.8409,Y 39.1174,Z 96,A 149.5819,B 24.9176,C -2.0965,E1 24.8554,E2 -64.419} C_DIS
LIN {X -82.3521,Y 42.1615,Z 96,A 147.4667,B 24.9171,C -2.1022,E1 24.858,E2 -62.306} C_DIS
LIN {X -80.8198,Y 45.0292,Z 96,A 145.4764,B 24.9166,C -2.1088,E1 24.8607,E2 -60.3209} C_DIS
LIN {X -79.3549,Y 47.5666,Z 96,A 143.4932,B 24.9166,C -2.1088,E1 24.8635,E2 -58.3276} C_DIS
LIN {X -77.5381,Y 50.4737,Z 96,A 141.3775,B 24.9161,C -2.115,E1 24.8667,E2 -56.2159} C_DIS
LIN {X -75.9168,Y 52.8782,Z 96,A 139.7181,B 24.9154,C -2.1241,E1 24.8692,E2 -54.5701} C_DIS
LIN {X -74.3075,Y 55.1196,Z 96,A 138.0385,B 24.9149,C -2.1296,E1 24.872,E2 -52.8954} C_DIS
LIN {X -72.5848,Y 57.3665,Z 96,A 136.1645,B 24.9149,C -2.1306,E1 24.8752,E2 -51.0149} C_DIS
LIN {X -70.4285,Y 59.994,Z 96,A 134.0461,B 24.9145,C -2.1357,E1 24.879,E2 -48.8987} C_DIS
LIN {X -68.1606,Y 62.5587,Z 96,A 131.9138,B 24.9141,C -2.1406,E1 24.883,E2 -46.7689} C_DIS
LIN {X -65.8181,Y 65.0188,Z 96,A 129.8004,B 24.9137,C -2.1455,E1 24.8871,E2 -44.6578} C_DIS
LIN {X -63.3866,Y 67.3914,Z 96,A 127.6838,B 24.9133,C -2.1501,E1 24.8913,E2 -42.5435} C_DIS
LIN {X -60.8496,Y 69.6906,Z 96,A 125.5519,B 24.9129,C -2.1545,E1 24.8958,E2 -40.4138} C_DIS
LIN {X -58.2494,Y 71.8781,Z 96,A 123.4396,B 24.9126,C -2.1589,E1 24.9003,E2 -38.3038} C_DIS
LIN {X -55.5809,Y 73.961,Z 96,A 121.309,B 24.9123,C -2.1623,E1 24.905,E2 -36.1735} C_DIS
LIN {X -52.8223,Y 75.9557,Z 96,A 119.2101,B 24.9119,C -2.1668,E1 24.9098,E2 -34.0781} C_DIS
LIN {X -50.0437,Y 77.8145,Z 96,A 117.1957,B 24.9115,C -2.1726,E1 24.9145,E2 -32.0707} C_DIS
LIN {X -47.5652,Y 79.3557,Z 96,A 115.2308,B 24.9116,C -2.1709,E1 24.9192,E2 -30.0959} C_DIS
LIN {X -45.0255,Y 80.8219,Z 96,A 113.4869,B 24.9112,C -2.1764,E1 24.9234,E2 -28.3599} C_DIS
LIN {X -42.1313,Y 82.3675,Z 96,A 111.4313,B 24.9109,C -2.179,E1 24.9285,E2 -26.3049} C_DIS
LIN {X -39.1056,Y 83.8464,Z 96,A 109.3416,B 24.9107,C -2.1822,E1 24.9338,E2 -24.2173} C_DIS
LIN {X -35.8994,Y 85.2683,Z 96,A 107.1887,B 24.9104,C -2.1859,E1 24.9393,E2 -22.0683} C_DIS
LIN {X -33.2874,Y 86.3233,Z 96,A 105.3523,B 24.9104,C -2.1853,E1 24.944,E2 -20.2266} C_DIS
LIN {X -30.5479,Y 87.3287,Z 96,A 103.7326,B 24.9097,C -2.1936,E1 24.9483,E2 -18.6234} C_DIS
LIN {X -28.3997,Y 88.0507,Z 96,A 102.216,B 24.9099,C -2.1917,E1 24.9523,E2 -17.0993} C_DIS
LIN {X -25.2677,Y 89,Z 96,A 100.1564,B 24.9099,C -2.1928,E1 24.9578,E2 -15.0391} C_DIS
LIN {X -21.9976,Y 89.8642,Z 96,A 98.0778,B 24.9096,C -2.1954,E1 24.9634,E2 -12.9636} C_DIS
LIN {X -18.6421,Y 90.6197,Z 96,A 95.9239,B 24.9096,C -2.1965,E1 24.9693,E2 -10.8096} C_DIS
LIN {X -15.3268,Y 91.239,Z 96,A 93.9217,B 24.9091,C -2.2009,E1 24.9748,E2 -8.8158} C_DIS
LIN {X -12.871,Y 91.6178,Z 96,A 92.3404,B 24.9091,C -2.2005,E1 24.9792,E2 -7.2323} C_DIS
LIN {X -9.5281,Y 92.0255,Z 96,A 90.2581,B 24.9091,C -2.2018,E1 24.9849,E2 -5.1517} C_DIS
LIN {X -6.3343,Y 92.3003,Z 96,A 88.2136,B 24.9091,C -2.2007,E1 24.9906,E2 -3.1038} C_DIS
LIN {X -2.7967,Y 92.4751,Z 96,A 86.0677,B 24.909,C -2.203,E1 24.9966,E2 -0.9629} C_DIS
LIN {X 0.5536,Y 92.5157,Z 96,A 83.9852,B 24.909,C -2.2032,E1 25.0024,E2 1.1192} C_DIS
LIN {X 3.4161,Y 92.4559,Z 96,A 82.1148,B 24.9092,C -2.2001,E1 25.0077,E2 2.9965} C_DIS
LIN {X 6.3308,Y 92.3005,Z 96,A 80.4155,B 24.9089,C -2.2038,E1 25.0124,E2 4.6864} C_DIS
LIN {X 9.5481,Y 92.0234,Z 96,A 78.4496,B 24.9089,C -2.2047,E1 25.0178,E2 6.649} C_DIS
LIN {X 12.4468,Y 91.678,Z 96,A 76.4871,B 24.9093,C -2.1991,E1 25.0233,E2 8.6232} C_DIS
LIN {X 15.8378,Y 91.1533,Z 96,A 74.337,B 24.9094,C -2.1975,E1 25.0292,E2 10.7748} C_DIS
LIN {X 19.1593,Y 90.5135,Z 96,A 72.2775,B 24.9094,C -2.1978,E1 25.0349,E2 12.8312} C_DIS
LIN {X 22.352,Y 89.7777,Z 96,A 70.2419,B 24.9095,C -2.1965,E1 25.0404,E2 14.867} C_DIS
LIN {X 25.3018,Y 88.9903,Z 96,A 68.5607,B 24.909,C -2.2023,E1 25.0449,E2 16.5315} C_DIS
LIN {X 27.9514,Y 88.1957,Z 96,A 66.8509,B 24.9091,C -2.2011,E1 25.0494,E2 18.2411} C_DIS
LIN {X 30.5573,Y 87.3254,Z 96,A 65.1031,B 24.9094,C -2.1981,E1 25.0541,E2 19.9927} C_DIS
LIN {X 32.8475,Y 86.4899,Z 96,A 63.6171,B 24.9094,C -2.1975,E1 25.0579,E2 21.4769} C_DIS
LIN {X 35.4355,Y 85.4639,Z 96,A 61.6997,B 24.9101,C -2.1891,E1 25.0629,E2 23.4099} C_DIS
LIN {X 38.5326,Y 84.1131,Z 96,A 59.6476,B 24.9101,C -2.1881,E1 25.0682,E2 25.4592} C_DIS
LIN {X 41.1786,Y 82.848,Z 96,A 58.0258,B 24.9098,C -2.1926,E1 25.0722,E2 27.066} C_DIS
LIN {X 43.6204,Y 81.5906,Z 96,A 56.138,B 24.9105,C -2.1839,E1 25.0769,E2 28.9693} C_DIS
LIN {X 46.1712,Y 80.1729,Z 96,A 54.4461,B 24.9105,C -2.1854,E1 25.081,E2 30.6525} C_DIS
LIN {X 48.5321,Y 78.7681,Z 96,A 52.8317,B 24.9104,C -2.1859,E1 25.0848,E2 32.2608} C_DIS
LIN {X 50.4467,Y 77.5558,Z 96,A 51.2044,B 24.9112,C -2.1758,E1 25.0887,E2 33.9066} C_DIS
LIN {X 53.2758,Y 75.6404,Z 96,A 49.1308,B 24.9114,C -2.1738,E1 25.0935,E2 35.9779} C_DIS
LIN {X 55.6382,Y 73.9179,Z 96,A 47.4399,B 24.9113,C -2.1749,E1 25.0972,E2 37.6602} C_DIS
LIN {X 58.2534,Y 71.8749,Z 96,A 45.3653,B 24.9116,C -2.1704,E1 25.1018,E2 39.7376} C_DIS
LIN {X 60.8727,Y 69.6705,Z 96,A 43.2528,B 24.912,C -2.1666,E1 25.1063,E2 41.851} C_DIS
LIN {X 63.387,Y 67.391,Z 96,A 41.1633,B 24.9123,C -2.1627,E1 25.1106,E2 43.9411} C_DIS
LIN {X 65.8169,Y 65.02,Z 96,A 39.0692,B 24.9126,C -2.1586,E1 25.1147,E2 46.0361} C_DIS
LIN {X 68.1703,Y 62.5482,Z 96,A 36.9662,B 24.913,C -2.1543,E1 25.1187,E2 48.1401} C_DIS
LIN {X 70.4238,Y 59.9996,Z 96,A 34.8656,B 24.9133,C -2.1497,E1 25.1226,E2 50.242} C_DIS
LIN {X 72.5852,Y 57.3659,Z 96,A 32.8064,B 24.9136,C -2.1465,E1 25.1262,E2 52.2991} C_DIS
LIN {X 74.4237,Y 54.961,Z 96,A 30.8621,B 24.9142,C -2.1394,E1 25.1295,E2 54.2509} C_DIS
LIN {X 76.297,Y 52.331,Z 96,A 29.026,B 24.9141,C -2.1403,E1 25.1324,E2 56.076} C_DIS
LIN {X 77.8151,Y 50.0427,Z 96,A 27.2856,B 24.9145,C -2.1345,E1 25.1351,E2 57.8214} C_DIS
LIN {X 79.106,Y 47.9762,Z 96,A 25.7514,B 24.9149,C -2.1296,E1 25.1373,E2 59.3594} C_DIS
LIN {X 81.0999,Y 44.5252,Z 96,A 23.1479,B 24.9159,C -2.1181,E1 25.1409,E2 61.9767} C_DIS
LIN {X 82.6726,Y 41.5324,Z 96,A 21.1069,B 24.9162,C -2.1142,E1 25.1435,E2 64.0159} C_DIS
LIN {X 84.1203,Y 38.5169,Z 96,A 19.2404,B 24.916,C -2.1158,E1 25.1457,E2 65.8685} C_DIS
LIN {X 85.0381,Y 36.4457,Z 96,A 17.654,B 24.9169,C -2.1051,E1 25.1475,E2 67.4716} C_DIS
LIN {X 86.1435,Y 33.7457,Z 96,A 15.9679,B 24.9169,C -2.1043,E1 25.1492,E2 69.1503} C_DIS
LIN {X 87.3387,Y 30.5192,Z 96,A 13.8474,B 24.9174,C -2.0984,E1 25.1513,E2 71.2728} C_DIS
LIN {X 88.3969,Y 27.3029,Z 96,A 11.7209,B 24.918,C -2.091,E1 25.1531,E2 73.4046} C_DIS
LIN {X 89.3376,Y 24.047,Z 96,A 9.6825,B 24.9183,C -2.0869,E1 25.1546,E2 75.4412} C_DIS
LIN {X 90.1583,Y 20.7593,Z 96,A 7.6387,B 24.9187,C -2.0824,E1 25.156,E2 77.4836} C_DIS
LIN {X 90.7409,Y 18.0516,Z 96,A 5.9755,B 24.9189,C -2.079,E1 25.1569,E2 79.1452} C_DIS
LIN {X 91.156,Y 15.8227,Z 96,A 4.3709,B 24.9199,C -2.0672,E1 25.1577,E2 80.7682} C_DIS
LIN {X 91.6508,Y 12.6386,Z 96,A 2.3857,B 24.9203,C -2.0613,E1 25.1585,E2 82.7556} C_DIS
LIN {X 92.0234,Y 9.5474,Z 96,A 0.6025,B 24.9203,C -2.0606,E1 25.159,E2 84.53} C_DIS
LIN {X 92.3006,Y 6.3301,Z 96,A -1.3508,B 24.9207,C -2.0559,E1 25.1595,E2 86.4827} C_DIS
LIN {X 92.453,Y 3.4838,Z 96,A -3.2638,B 24.9216,C -2.0448,E1 25.1597,E2 88.4106} C_DIS
LIN {X 92.5187,Y 0.1036,Z 96,A -5.1492,B 24.9216,C -2.0458,E1 25.1597,E2 90.2825} C_DIS
LIN {X 92.4913,Y -2.2666,Z 96,A -6.5918,B 24.9218,C -2.042,E1 25.1597,E2 91.7255} C_DIS
LIN {X 92.3815,Y -5.0125,Z 96,A -8.3307,B 24.9223,C -2.0352,E1 25.1595,E2 93.4701} C_DIS
LIN {X 92.1816,Y -7.8913,Z 96,A -10.2523,B 24.9232,C -2.0244,E1 25.1591,E2 95.4057} C_DIS
Enddeposition()
END
